LIN {X 0,Y 197.499,Z 678.187,A -85,B 0,C 180,E1 -21855.576,E2 -21855.576} C_VEL
LIN {X 0,Y 195.78,Z 682.074,A -85,B 0,C 180,E1 -21858.613,E2 -21858.613} C_VEL
LIN {X 0,Y 194.459,Z 684.943,A -85,B 0,C 180,E1 -21861.688,E2 -21861.688} C_VEL
LIN {X 0,Y 194.056,Z 686.281,A -85,B 0,C 180,E1 -21863.763,E2 -21863.763} C_VEL
LIN {X 0,Y 193.799,Z 687.228,A -85,B 0,C 180,E1 -21865.841,E2 -21865.841} C_VEL
LIN {X 0,Y 193.417,Z 688.055,A -85,B 0,C 180,E1 -21870,E2 -21870} C_VEL
LIN {X 0,Y 193.796,Z 687.282,A -85,B 0,C 180,E1 -21874.159,E2 -21874.159} C_VEL
LIN {X 0,Y 194.443,Z 685.054,A -85,B 0,C 180,E1 -21878.313,E2 -21878.313} C_VEL
LIN {X 0,Y 195.772,Z 682.224,A -85,B 0,C 180,E1 -21881.387,E2 -21881.387} C_VEL
LIN {X 0,Y 197.474,Z 678.391,A -85,B 0,C 180,E1 -21884.425,E2 -21884.425} C_VEL
LIN {X 0,Y 199.366,Z 673.305,A -85,B 0,C 180,E1 -21887.541,E2 -21887.541} C_VEL
LIN {X 0,Y 201.662,Z 667.266,A -85,B 0,C 180,E1 -21890.395,E2 -21890.395} C_VEL
LIN {X 0,Y 204.413,Z 659.477,A -85,B 0,C 180,E1 -21893.289,E2 -21893.289} C_VEL
LIN {X 0,Y 207.374,Z 649.797,A -85,B 0,C 180,E1 -21896.14,E2 -21896.14} C_VEL
LIN {X 0,Y 209.903,Z 640.74,A -85,B 0,C 180,E1 -21898.224,E2 -21898.224} C_VEL
LIN {X 0,Y 212.551,Z 630.212,A -85,B 0,C 180,E1 -21900.13,E2 -21900.13} C_VEL
LIN {X 0,Y 214.851,Z 618.67,A -85,B 0,C 180,E1 -21901.781,E2 -21901.781} C_VEL
LIN {X 0,Y 216.718,Z 607.358,A -85,B 0,C 180,E1 -21902.997,E2 -21902.997} C_VEL
LIN {X 0,Y 217.85,Z 594.616,A -85,B 0,C 180,E1 -21904.049,E2 -21904.049} C_VEL
LIN {X 0,Y 218.527,Z 581.541,A -85,B 0,C 180,E1 -21904.74,E2 -21904.74} C_VEL
LIN {X 0,Y 219.472,Z 546.637,A -85,B 0,C 180,E1 -21905.962,E2 -21905.962} C_VEL
LIN {X 0,Y 212.575,Z 532.953,A -85,B 0,C 180,E1 -21907.952,E2 -21907.952} C_VEL
LIN {X 0,Y 205.517,Z 520.799,A -85,B 0,C 180,E1 -21910.109,E2 -21910.109} C_VEL
LIN {X 0,Y 200.207,Z 512.651,A -85,B 0,C 180,E1 -21911.836,E2 -21911.836} C_VEL
LIN {X 0,Y 197.755,Z 509.046,A -85,B 0,C 180,E1 -21912.674,E2 -21912.674} C_VEL
LIN {X 0,Y 195.601,Z 505.666,A -85,B 0,C 180,E1 -21913.449,E2 -21913.449} C_VEL
LIN {X 0,Y 193.302,Z 502.912,A -85,B 0,C 180,E1 -21914.263,E2 -21914.263} C_VEL
LIN {X 0,Y 192.631,Z 500.948,A -85,B 0,C 180,E1 -21914.75,E2 -21914.75} C_VEL
LIN {X 0,Y 192.52,Z 500.498,A -85,B 0,C 180,E1 -21915.59,E2 -21915.59} C_VEL
LIN {X 0,Y 192.507,Z 500.453,A -85,B 0,C 180,E1 -21920.053,E2 -21920.053} C_VEL
LIN {X 0,Y 192.558,Z 500.5,A -85,B 0,C 180,E1 -21924.27,E2 -21924.27} C_VEL
LIN {X 0,Y 192.605,Z 500.44,A -85,B 0,C 180,E1 -21927.059,E2 -21927.059} C_VEL
LIN {X 0,Y 192.658,Z 500.435,A -85,B 0,C 180,E1 -21931.691,E2 -21931.691} C_VEL
LIN {X 0,Y 192.682,Z 500.469,A -85,B 0,C 180,E1 -21936.345,E2 -21936.345} C_VEL
LIN {X 0,Y 192.728,Z 500.474,A -85,B 0,C 180,E1 -21941.458,E2 -21941.458} C_VEL
LIN {X 0,Y 192.848,Z 500.463,A -85,B 0,C 180,E1 -21947.37,E2 -21947.37} C_VEL
LIN {X 0,Y 193.064,Z 500.413,A -85,B 0,C 180,E1 -21951.627,E2 -21951.627} C_VEL
LIN {X 0,Y 193.259,Z 500.383,A -85,B 0,C 180,E1 -21957.916,E2 -21957.916} C_VEL
LIN {X 0,Y 193.442,Z 500.381,A -85,B 0,C 180,E1 -21960,E2 -21960} C_VEL
LIN {X 0,Y 192.968,Z 500.419,A -85,B 0,C 180,E1 -21964.177,E2 -21964.177} C_VEL
LIN {X 0,Y 193.032,Z 500.437,A -85,B 0,C 180,E1 -21968.374,E2 -21968.374} C_VEL
LIN {X 0,Y 192.798,Z 500.454,A -85,B 0,C 180,E1 -21972.634,E2 -21972.634} C_VEL
LIN {X 0,Y 192.754,Z 500.439,A -85,B 0,C 180,E1 -21976.959,E2 -21976.959} C_VEL
LIN {X 0,Y 192.626,Z 500.465,A -85,B 0,C 180,E1 -21981.398,E2 -21981.398} C_VEL
LIN {X 0,Y 192.661,Z 500.476,A -85,B 0,C 180,E1 -21984.225,E2 -21984.225} C_VEL
LIN {X 0,Y 192.647,Z 500.468,A -85,B 0,C 180,E1 -21988.893,E2 -21988.893} C_VEL
LIN {X 0,Y 192.596,Z 500.469,A -85,B 0,C 180,E1 -21993.186,E2 -21993.186} C_VEL
LIN {X 0,Y 192.61,Z 500.721,A -85,B 0,C 180,E1 -21994.759,E2 -21994.759} C_VEL
LIN {X 0,Y 195.27,Z 509.211,A -85,B 0,C 180,E1 -21999.706,E2 -21999.706} C_VEL
LIN {X 0,Y 197.737,Z 517.882,A -85,B 0,C 180,E1 -22004.176,E2 -22004.176} C_VEL
LIN {X 0,Y 198.984,Z 522.474,A -85,B 0,C 180,E1 -22006.298,E2 -22006.298} C_VEL
LIN {X 0,Y 204.591,Z 534.212,A -85,B 0,C 180,E1 -22008.344,E2 -22008.344} C_VEL
LIN {X 0,Y 210.617,Z 548.053,A -85,B 0,C 180,E1 -22010.333,E2 -22010.333} C_VEL
LIN {X 0,Y 211.524,Z 550.943,A -85,B 0,C 180,E1 -22010.653,E2 -22010.653} C_VEL
LIN {X 0,Y 214.13,Z 576.298,A -85,B 0,C 180,E1 -22012.25,E2 -22012.25} C_VEL
LIN {X 0,Y 216.129,Z 604.791,A -85,B 0,C 180,E1 -22013.789,E2 -22013.789} C_VEL
LIN {X 0,Y 216.582,Z 612.878,A -85,B 0,C 180,E1 -22014.194,E2 -22014.194} C_VEL
LIN {X 0,Y 216.05,Z 618.711,A -85,B 0,C 180,E1 -22014.32,E2 -22014.32} C_VEL
LIN {X 0,Y 214.533,Z 624.449,A -85,B 0,C 180,E1 -22014.265,E2 -22014.265} C_VEL
LIN {X 0,Y 209.975,Z 637.636,A -85,B 0,C 180,E1 -22014.06,E2 -22014.06} C_VEL
LIN {X 0,Y 208.782,Z 643.411,A -85,B 0,C 180,E1 -22014.266,E2 -22014.266} C_VEL
LIN {X 0,Y 206.963,Z 656.057,A -85,B 0,C 180,E1 -22015.187,E2 -22015.187} C_VEL
LIN {X 0,Y 205.094,Z 665.781,A -85,B 0,C 180,E1 -22016.163,E2 -22016.163} C_VEL
LIN {X 0,Y 202.171,Z 677.646,A -85,B 0,C 180,E1 -22017.693,E2 -22017.693} C_VEL
LIN {X 0,Y 198.651,Z 689.501,A -85,B 0,C 180,E1 -22019.726,E2 -22019.726} C_VEL
LIN {X 0,Y 195.192,Z 700.074,A -85,B 0,C 180,E1 -22022.092,E2 -22022.092} C_VEL
LIN {X 0,Y 192.203,Z 708.672,A -85,B 0,C 180,E1 -22024.556,E2 -22024.556} C_VEL
LIN {X 0,Y 189.306,Z 717.125,A -85,B 0,C 180,E1 -22027.634,E2 -22027.634} C_VEL
LIN {X 0,Y 186.845,Z 723.957,A -85,B 0,C 180,E1 -22030.785,E2 -22030.785} C_VEL
LIN {X 0,Y 185.18,Z 730.323,A -85,B 0,C 180,E1 -22034.594,E2 -22034.594} C_VEL
LIN {X 0,Y 184.386,Z 734.512,A -85,B 0,C 180,E1 -22037.899,E2 -22037.899} C_VEL
LIN {X 0,Y 184.257,Z 737.676,A -85,B 0,C 180,E1 -22041.224,E2 -22041.224} C_VEL
LIN {X 0,Y 184.433,Z 739.217,A -85,B 0,C 180,E1 -22043.436,E2 -22043.436} C_VEL
LIN {X 0,Y 184.793,Z 740.348,A -85,B 0,C 180,E1 -22045.638,E2 -22045.638} C_VEL
LIN {X 0,Y 185.84,Z 741.38,A -85,B 0,C 180,E1 -22050,E2 -22050} C_VEL
LIN {X 0,Y 184.812,Z 740.331,A -85,B 0,C 180,E1 -22054.362,E2 -22054.362} C_VEL
LIN {X 0,Y 184.36,Z 738.485,A -85,B 0,C 180,E1 -22057.629,E2 -22057.629} C_VEL
LIN {X 0,Y 184.285,Z 735.608,A -85,B 0,C 180,E1 -22060.992,E2 -22060.992} C_VEL
LIN {X 0,Y 184.851,Z 731.751,A -85,B 0,C 180,E1 -22064.307,E2 -22064.307} C_VEL
LIN {X 0,Y 186.073,Z 726.793,A -85,B 0,C 180,E1 -22067.587,E2 -22067.587} C_VEL
LIN {X 0,Y 188.212,Z 720.14,A -85,B 0,C 180,E1 -22071.009,E2 -22071.009} C_VEL
LIN {X 0,Y 190.673,Z 712.967,A -85,B 0,C 180,E1 -22073.919,E2 -22073.919} C_VEL
LIN {X 0,Y 193.385,Z 705.23,A -85,B 0,C 180,E1 -22076.435,E2 -22076.435} C_VEL
LIN {X 0,Y 196.501,Z 695.896,A -85,B 0,C 180,E1 -22078.87,E2 -22078.87} C_VEL
LIN {X 0,Y 199.834,Z 685.58,A -85,B 0,C 180,E1 -22080.953,E2 -22080.953} C_VEL
LIN {X 0,Y 203.037,Z 674.165,A -85,B 0,C 180,E1 -22082.741,E2 -22082.741} C_VEL
LIN {X 0,Y 205.619,Z 662.301,A -85,B 0,C 180,E1 -22084.181,E2 -22084.181} C_VEL
LIN {X 0,Y 207.884,Z 649.433,A -85,B 0,C 180,E1 -22085.29,E2 -22085.29} C_VEL
LIN {X 0,Y 209.429,Z 635.954,A -85,B 0,C 180,E1 -22086.076,E2 -22086.076} C_VEL
LIN {X 0,Y 210.609,Z 611.893,A -85,B 0,C 180,E1 -22086.916,E2 -22086.916} C_VEL
LIN {X 0,Y 208.307,Z 576.822,A -85,B 0,C 180,E1 -22088.861,E2 -22088.861} C_VEL
LIN {X 0,Y 205.939,Z 552.664,A -85,B 0,C 180,E1 -22090.435,E2 -22090.435} C_VEL
LIN {X 0,Y 201.062,Z 541.037,A -85,B 0,C 180,E1 -22092.124,E2 -22092.124} C_VEL
LIN {X 0,Y 196.044,Z 530.426,A -85,B 0,C 180,E1 -22093.935,E2 -22093.935} C_VEL
LIN {X 0,Y 193.42,Z 525.344,A -85,B 0,C 180,E1 -22094.918,E2 -22094.918} C_VEL
LIN {X 0,Y 191.371,Z 520.955,A -85,B 0,C 180,E1 -22095.844,E2 -22095.844} C_VEL
LIN {X 0,Y 189.045,Z 512.792,A -85,B 0,C 180,E1 -22100.112,E2 -22100.112} C_VEL
LIN {X 0,Y 186.806,Z 505.66,A -85,B 0,C 180,E1 -22104.328,E2 -22104.328} C_VEL
LIN {X 0,Y 185.567,Z 501.428,A -85,B 0,C 180,E1 -22107.137,E2 -22107.137} C_VEL
LIN {X 0,Y 185.579,Z 501.355,A -85,B 0,C 180,E1 -22110.575,E2 -22110.575} C_VEL
LIN {X 0,Y 185.584,Z 501.35,A -85,B 0,C 180,E1 -22115.382,E2 -22115.382} C_VEL
LIN {X 0,Y 185.67,Z 501.308,A -85,B 0,C 180,E1 -22121.134,E2 -22121.134} C_VEL
LIN {X 0,Y 185.691,Z 501.349,A -85,B 0,C 180,E1 -22124.637,E2 -22124.637} C_VEL
LIN {X 0,Y 185.885,Z 501.307,A -85,B 0,C 180,E1 -22129.418,E2 -22129.418} C_VEL
LIN {X 0,Y 185.944,Z 501.313,A -85,B 0,C 180,E1 -22133.489,E2 -22133.489} C_VEL
LIN {X 0,Y 186.202,Z 501.28,A -85,B 0,C 180,E1 -22137.837,E2 -22137.837} C_VEL
LIN {X 0,Y 186.405,Z 501.261,A -85,B 0,C 180,E1 -22140,E2 -22140} C_VEL
LIN {X 0,Y 185.916,Z 501.309,A -85,B 0,C 180,E1 -22144.336,E2 -22144.336} C_VEL
LIN {X 0,Y 185.979,Z 501.293,A -85,B 0,C 180,E1 -22148.694,E2 -22148.694} C_VEL
LIN {X 0,Y 185.724,Z 501.35,A -85,B 0,C 180,E1 -22153.123,E2 -22153.123} C_VEL
LIN {X 0,Y 185.685,Z 501.339,A -85,B 0,C 180,E1 -22157.626,E2 -22157.626} C_VEL
LIN {X 0,Y 185.577,Z 501.347,A -85,B 0,C 180,E1 -22162.254,E2 -22162.254} C_VEL
LIN {X 0,Y 185.556,Z 501.345,A -85,B 0,C 180,E1 -22167.033,E2 -22167.033} C_VEL
LIN {X 0,Y 185.575,Z 501.3,A -85,B 0,C 180,E1 -22169.494,E2 -22169.494} C_VEL
LIN {X 0,Y 185.496,Z 501.359,A -85,B 0,C 180,E1 -22174.633,E2 -22174.633} C_VEL
LIN {X 0,Y 185.499,Z 501.35,A -85,B 0,C 180,E1 -22177.315,E2 -22177.315} C_VEL
LIN {X 0,Y 185.469,Z 501.445,A -85,B 0,C 180,E1 -22182.771,E2 -22182.771} C_VEL
LIN {X 0,Y 185.629,Z 502.258,A -85,B 0,C 180,E1 -22183.39,E2 -22183.39} C_VEL
LIN {X 0,Y 187.124,Z 505.129,A -85,B 0,C 180,E1 -22184.12,E2 -22184.12} C_VEL
LIN {X 0,Y 188.874,Z 506.941,A -85,B 0,C 180,E1 -22184.781,E2 -22184.781} C_VEL
LIN {X 0,Y 190.87,Z 510.07,A -85,B 0,C 180,E1 -22185.568,E2 -22185.568} C_VEL
LIN {X 0,Y 192.372,Z 512.165,A -85,B 0,C 180,E1 -22186.129,E2 -22186.129} C_VEL
LIN {X 0,Y 197.664,Z 519.995,A -85,B 0,C 180,E1 -22188.019,E2 -22188.019} C_VEL
LIN {X 0,Y 203.928,Z 530.25,A -85,B 0,C 180,E1 -22190.108,E2 -22190.108} C_VEL
LIN {X 0,Y 211.258,Z 543.831,A -85,B 0,C 180,E1 -22192.39,E2 -22192.39} C_VEL
LIN {X 0,Y 213.706,Z 549.024,A -85,B 0,C 180,E1 -22193.13,E2 -22193.13} C_VEL
LIN {X 0,Y 212.454,Z 587.486,A -85,B 0,C 180,E1 -22194.541,E2 -22194.541} C_VEL
LIN {X 0,Y 211.413,Z 601.314,A -85,B 0,C 180,E1 -22195.451,E2 -22195.451} C_VEL
LIN {X 0,Y 209.843,Z 613.54,A -85,B 0,C 180,E1 -22196.614,E2 -22196.614} C_VEL
LIN {X 0,Y 207.843,Z 624.696,A -85,B 0,C 180,E1 -22198.032,E2 -22198.032} C_VEL
LIN {X 0,Y 205.358,Z 635.064,A -85,B 0,C 180,E1 -22199.683,E2 -22199.683} C_VEL
LIN {X 0,Y 202.579,Z 645.376,A -85,B 0,C 180,E1 -22201.792,E2 -22201.792} C_VEL
LIN {X 0,Y 200.031,Z 653.784,A -85,B 0,C 180,E1 -22203.949,E2 -22203.949} C_VEL
LIN {X 0,Y 197.499,Z 661.508,A -85,B 0,C 180,E1 -22206.402,E2 -22206.402} C_VEL
LIN {X 0,Y 194.636,Z 669.172,A -85,B 0,C 180,E1 -22209.443,E2 -22209.443} C_VEL
LIN {X 0,Y 191.978,Z 675.971,A -85,B 0,C 180,E1 -22212.971,E2 -22212.971} C_VEL
LIN {X 0,Y 190.005,Z 680.577,A -85,B 0,C 180,E1 -22216.089,E2 -22216.089} C_VEL
LIN {X 0,Y 188.343,Z 684.112,A -85,B 0,C 180,E1 -22219.247,E2 -22219.247} C_VEL
LIN {X 0,Y 187.506,Z 685.933,A -85,B 0,C 180,E1 -22221.378,E2 -22221.378} C_VEL
LIN {X 0,Y 187.07,Z 687.27,A -85,B 0,C 180,E1 -22223.529,E2 -22223.529} C_VEL
LIN {X 0,Y 186.791,Z 688.216,A -85,B 0,C 180,E1 -22225.685,E2 -22225.685} C_VEL
LIN {X 0,Y 186.389,Z 689.043,A -85,B 0,C 180,E1 -22230,E2 -22230} C_VEL
LIN {X 0,Y 186.788,Z 688.269,A -85,B 0,C 180,E1 -22234.316,E2 -22234.316} C_VEL
LIN {X 0,Y 187.489,Z 686.042,A -85,B 0,C 180,E1 -22238.623,E2 -22238.623} C_VEL
LIN {X 0,Y 188.888,Z 683.211,A -85,B 0,C 180,E1 -22241.808,E2 -22241.808} C_VEL
LIN {X 0,Y 190.676,Z 679.378,A -85,B 0,C 180,E1 -22244.952,E2 -22244.952} C_VEL
LIN {X 0,Y 192.676,Z 674.291,A -85,B 0,C 180,E1 -22248.171,E2 -22248.171} C_VEL
LIN {X 0,Y 195.09,Z 668.252,A -85,B 0,C 180,E1 -22251.115,E2 -22251.115} C_VEL
LIN {X 0,Y 197.977,Z 660.463,A -85,B 0,C 180,E1 -22254.094,E2 -22254.094} C_VEL
LIN {X 0,Y 201.088,Z 650.782,A -85,B 0,C 180,E1 -22257.022,E2 -22257.022} C_VEL
LIN {X 0,Y 203.74,Z 641.724,A -85,B 0,C 180,E1 -22259.159,E2 -22259.159} C_VEL
LIN {X 0,Y 206.51,Z 631.193,A -85,B 0,C 180,E1 -22261.107,E2 -22261.107} C_VEL
LIN {X 0,Y 208.95,Z 619.496,A -85,B 0,C 180,E1 -22262.815,E2 -22262.815} C_VEL
LIN {X 0,Y 210.905,Z 607.994,A -85,B 0,C 180,E1 -22264.071,E2 -22264.071} C_VEL
LIN {X 0,Y 212.098,Z 595.07,A -85,B 0,C 180,E1 -22265.148,E2 -22265.148} C_VEL
LIN {X 0,Y 212.79,Z 581.576,A -85,B 0,C 180,E1 -22265.865,E2 -22265.865} C_VEL
LIN {X 0,Y 213.713,Z 548.894,A -85,B 0,C 180,E1 -22267.038,E2 -22267.038} C_VEL
LIN {X 0,Y 207.503,Z 536.628,A -85,B 0,C 180,E1 -22268.93,E2 -22268.93} C_VEL
LIN {X 0,Y 201.238,Z 525.581,A -85,B 0,C 180,E1 -22270.954,E2 -22270.954} C_VEL
LIN {X 0,Y 194.118,Z 514.597,A -85,B 0,C 180,E1 -22273.425,E2 -22273.425} C_VEL
LIN {X 0,Y 190.785,Z 509.938,A -85,B 0,C 180,E1 -22274.658,E2 -22274.658} C_VEL
LIN {X 0,Y 188.759,Z 506.737,A -85,B 0,C 180,E1 -22275.463,E2 -22275.463} C_VEL
LIN {X 0,Y 186.229,Z 503.818,A -85,B 0,C 180,E1 -22276.45,E2 -22276.45} C_VEL
LIN {X 0,Y 185.573,Z 501.969,A -85,B 0,C 180,E1 -22276.928,E2 -22276.928} C_VEL
LIN {X 0,Y 185.46,Z 501.409,A -85,B 0,C 180,E1 -22277.617,E2 -22277.617} C_VEL
LIN {X 0,Y 185.5,Z 501.349,A -85,B 0,C 180,E1 -22282.712,E2 -22282.712} C_VEL
LIN {X 0,Y 185.539,Z 501.306,A -85,B 0,C 180,E1 -22287.974,E2 -22287.974} C_VEL
LIN {X 0,Y 185.578,Z 501.301,A -85,B 0,C 180,E1 -22290.576,E2 -22290.576} C_VEL
LIN {X 0,Y 185.577,Z 501.365,A -85,B 0,C 180,E1 -22295.381,E2 -22295.381} C_VEL
LIN {X 0,Y 185.671,Z 501.356,A -85,B 0,C 180,E1 -22301.134,E2 -22301.134} C_VEL
LIN {X 0,Y 185.759,Z 501.346,A -85,B 0,C 180,E1 -22306.879,E2 -22306.879} C_VEL
LIN {X 0,Y 186.01,Z 501.289,A -85,B 0,C 180,E1 -22311.307,E2 -22311.307} C_VEL
LIN {X 0,Y 186.203,Z 501.261,A -85,B 0,C 180,E1 -22317.837,E2 -22317.837} C_VEL
LIN {X 0,Y 186.405,Z 501.257,A -85,B 0,C 180,E1 -22320,E2 -22320} C_VEL
LIN {X 0,Y 185.915,Z 501.297,A -85,B 0,C 180,E1 -22324.336,E2 -22324.336} C_VEL
LIN {X 0,Y 185.979,Z 501.31,A -85,B 0,C 180,E1 -22328.694,E2 -22328.694} C_VEL
LIN {X 0,Y 185.725,Z 501.341,A -85,B 0,C 180,E1 -22333.123,E2 -22333.123} C_VEL
LIN {X 0,Y 185.686,Z 501.311,A -85,B 0,C 180,E1 -22337.625,E2 -22337.625} C_VEL
LIN {X 0,Y 185.59,Z 501.358,A -85,B 0,C 180,E1 -22342.252,E2 -22342.252} C_VEL
LIN {X 0,Y 185.559,Z 501.335,A -85,B 0,C 180,E1 -22347.033,E2 -22347.033} C_VEL
LIN {X 0,Y 185.576,Z 501.358,A -85,B 0,C 180,E1 -22349.494,E2 -22349.494} C_VEL
LIN {X 0,Y 185.603,Z 501.511,A -85,B 0,C 180,E1 -22352.888,E2 -22352.888} C_VEL
LIN {X 0,Y 188.362,Z 510.35,A -85,B 0,C 180,E1 -22358.417,E2 -22358.417} C_VEL
LIN {X 0,Y 190.741,Z 518.676,A -85,B 0,C 180,E1 -22362.975,E2 -22362.975} C_VEL
LIN {X 0,Y 191.435,Z 521.22,A -85,B 0,C 180,E1 -22364.138,E2 -22364.138} C_VEL
LIN {X 0,Y 195.498,Z 529.272,A -85,B 0,C 180,E1 -22365.767,E2 -22365.767} C_VEL
LIN {X 0,Y 200.116,Z 538.807,A -85,B 0,C 180,E1 -22367.449,E2 -22367.449} C_VEL
LIN {X 0,Y 205.59,Z 551.566,A -85,B 0,C 180,E1 -22369.358,E2 -22369.358} C_VEL
LIN {X 0,Y 206.205,Z 554.163,A -85,B 0,C 180,E1 -22369.615,E2 -22369.615} C_VEL
LIN {X 0,Y 208.646,Z 579.601,A -85,B 0,C 180,E1 -22371.257,E2 -22371.257} C_VEL
LIN {X 0,Y 210.719,Z 611.4,A -85,B 0,C 180,E1 -22373.016,E2 -22373.016} C_VEL
LIN {X 0,Y 209.623,Z 634.88,A -85,B 0,C 180,E1 -22373.824,E2 -22373.824} C_VEL
LIN {X 0,Y 208.782,Z 643.411,A -85,B 0,C 180,E1 -22374.266,E2 -22374.266} C_VEL
LIN {X 0,Y 207.502,Z 649.097,A -85,B 0,C 180,E1 -22374.532,E2 -22374.532} C_VEL
LIN {X 0,Y 203.648,Z 658.159,A -85,B 0,C 180,E1 -22374.851,E2 -22374.851} C_VEL
LIN {X 0,Y 199.388,Z 666.921,A -85,B 0,C 180,E1 -22375.368,E2 -22375.368} C_VEL
LIN {X 0,Y 197.488,Z 672.139,A -85,B 0,C 180,E1 -22375.949,E2 -22375.949} C_VEL
LIN {X 0,Y 194.138,Z 683.569,A -85,B 0,C 180,E1 -22377.727,E2 -22377.727} C_VEL
LIN {X 0,Y 190.672,Z 694.076,A -85,B 0,C 180,E1 -22379.855,E2 -22379.855} C_VEL
LIN {X 0,Y 187.618,Z 702.705,A -85,B 0,C 180,E1 -22382.081,E2 -22382.081} C_VEL
LIN {X 0,Y 184.689,Z 710.708,A -85,B 0,C 180,E1 -22384.654,E2 -22384.654} C_VEL
LIN {X 0,Y 181.809,Z 718.61,A -85,B 0,C 180,E1 -22387.876,E2 -22387.876} C_VEL
LIN {X 0,Y 179.783,Z 723.985,A -85,B 0,C 180,E1 -22390.593,E2 -22390.593} C_VEL
LIN {X 0,Y 178.284,Z 729.317,A -85,B 0,C 180,E1 -22393.982,E2 -22393.982} C_VEL
LIN {X 0,Y 177.383,Z 733.505,A -85,B 0,C 180,E1 -22397.414,E2 -22397.414} C_VEL
LIN {X 0,Y 177.203,Z 736.673,A -85,B 0,C 180,E1 -22400.872,E2 -22400.872} C_VEL
LIN {X 0,Y 177.356,Z 738.215,A -85,B 0,C 180,E1 -22403.173,E2 -22403.173} C_VEL
LIN {X 0,Y 177.703,Z 739.348,A -85,B 0,C 180,E1 -22405.463,E2 -22405.463} C_VEL
LIN {X 0,Y 178.789,Z 740.389,A -85,B 0,C 180,E1 -22410,E2 -22410} C_VEL
LIN {X 0,Y 177.721,Z 739.331,A -85,B 0,C 180,E1 -22414.536,E2 -22414.536} C_VEL
LIN {X 0,Y 177.286,Z 737.664,A -85,B 0,C 180,E1 -22417.67,E2 -22417.67} C_VEL
LIN {X 0,Y 177.265,Z 734.601,A -85,B 0,C 180,E1 -22421.433,E2 -22421.433} C_VEL
LIN {X 0,Y 177.906,Z 730.741,A -85,B 0,C 180,E1 -22424.878,E2 -22424.878} C_VEL
LIN {X 0,Y 179.241,Z 725.782,A -85,B 0,C 180,E1 -22428.281,E2 -22428.281} C_VEL
LIN {X 0,Y 181.37,Z 719.664,A -85,B 0,C 180,E1 -22431.567,E2 -22431.567} C_VEL
LIN {X 0,Y 184.153,Z 711.958,A -85,B 0,C 180,E1 -22434.822,E2 -22434.822} C_VEL
LIN {X 0,Y 187.016,Z 704.223,A -85,B 0,C 180,E1 -22437.409,E2 -22437.409} C_VEL
LIN {X 0,Y 190.307,Z 694.894,A -85,B 0,C 180,E1 -22439.903,E2 -22439.903} C_VEL
LIN {X 0,Y 193.787,Z 684.579,A -85,B 0,C 180,E1 -22442.032,E2 -22442.032} C_VEL
LIN {X 0,Y 197.099,Z 673.161,A -85,B 0,C 180,E1 -22443.858,E2 -22443.858} C_VEL
LIN {X 0,Y 199.741,Z 661.289,A -85,B 0,C 180,E1 -22445.334,E2 -22445.334} C_VEL
LIN {X 0,Y 202.108,Z 648.568,A -85,B 0,C 180,E1 -22446.443,E2 -22446.443} C_VEL
LIN {X 0,Y 203.614,Z 636.122,A -85,B 0,C 180,E1 -22447.197,E2 -22447.197} C_VEL
LIN {X 0,Y 204.903,Z 615.139,A -85,B 0,C 180,E1 -22447.94,E2 -22447.94} C_VEL
LIN {X 0,Y 203.278,Z 585.097,A -85,B 0,C 180,E1 -22449.603,E2 -22449.603} C_VEL
LIN {X 0,Y 200.708,Z 555.786,A -85,B 0,C 180,E1 -22451.529,E2 -22451.529} C_VEL
LIN {X 0,Y 197.732,Z 548.261,A -85,B 0,C 180,E1 -22452.627,E2 -22452.627} C_VEL
LIN {X 0,Y 192.465,Z 536.379,A -85,B 0,C 180,E1 -22454.633,E2 -22454.633} C_VEL
LIN {X 0,Y 188.757,Z 529.157,A -85,B 0,C 180,E1 -22456.095,E2 -22456.095} C_VEL
LIN {X 0,Y 186.274,Z 524.432,A -85,B 0,C 180,E1 -22457.123,E2 -22457.123} C_VEL
LIN {X 0,Y 183.734,Z 519.425,A -85,B 0,C 180,E1 -22458.348,E2 -22458.348} C_VEL
LIN {X 0,Y 181.965,Z 513.227,A -85,B 0,C 180,E1 -22461.832,E2 -22461.832} C_VEL
LIN {X 0,Y 179.496,Z 505.59,A -85,B 0,C 180,E1 -22466.759,E2 -22466.759} C_VEL
LIN {X 0,Y 178.49,Z 502.306,A -85,B 0,C 180,E1 -22469.211,E2 -22469.211} C_VEL
LIN {X 0,Y 178.503,Z 502.219,A -85,B 0,C 180,E1 -22474.336,E2 -22474.336} C_VEL
LIN {X 0,Y 178.526,Z 502.208,A -85,B 0,C 180,E1 -22479.249,E2 -22479.249} C_VEL
LIN {X 0,Y 178.646,Z 502.183,A -85,B 0,C 180,E1 -22481.656,E2 -22481.656} C_VEL
LIN {X 0,Y 178.654,Z 502.228,A -85,B 0,C 180,E1 -22486.348,E2 -22486.348} C_VEL
LIN {X 0,Y 178.908,Z 502.189,A -85,B 0,C 180,E1 -22490.96,E2 -22490.96} C_VEL
LIN {X 0,Y 179.148,Z 502.157,A -85,B 0,C 180,E1 -22497.752,E2 -22497.752} C_VEL
LIN {X 0,Y 179.368,Z 502.137,A -85,B 0,C 180,E1 -22500,E2 -22500} C_VEL
LIN {X 0,Y 178.864,Z 502.189,A -85,B 0,C 180,E1 -22504.507,E2 -22504.507} C_VEL
LIN {X 0,Y 178.908,Z 502.172,A -85,B 0,C 180,E1 -22509.041,E2 -22509.041} C_VEL
LIN {X 0,Y 178.652,Z 502.226,A -85,B 0,C 180,E1 -22513.653,E2 -22513.653} C_VEL
LIN {X 0,Y 178.619,Z 502.237,A -85,B 0,C 180,E1 -22519.215,E2 -22519.215} C_VEL
LIN {X 0,Y 178.517,Z 502.248,A -85,B 0,C 180,E1 -22525.115,E2 -22525.115} C_VEL
LIN {X 0,Y 178.519,Z 502.175,A -85,B 0,C 180,E1 -22529.993,E2 -22529.993} C_VEL
LIN {X 0,Y 178.482,Z 502.219,A -85,B 0,C 180,E1 -22534.22,E2 -22534.22} C_VEL
LIN {X 0,Y 178.449,Z 502.268,A -85,B 0,C 180,E1 -22540.159,E2 -22540.159} C_VEL
LIN {X 0,Y 178.595,Z 503.083,A -85,B 0,C 180,E1 -22540.898,E2 -22540.898} C_VEL
LIN {X 0,Y 179.978,Z 505.859,A -85,B 0,C 180,E1 -22541.674,E2 -22541.674} C_VEL
LIN {X 0,Y 181.907,Z 507.76,A -85,B 0,C 180,E1 -22542.488,E2 -22542.488} C_VEL
LIN {X 0,Y 183.903,Z 510.97,A -85,B 0,C 180,E1 -22543.369,E2 -22543.369} C_VEL
LIN {X 0,Y 185.419,Z 512.873,A -85,B 0,C 180,E1 -22543.986,E2 -22543.986} C_VEL
LIN {X 0,Y 189.076,Z 518.203,A -85,B 0,C 180,E1 -22545.447,E2 -22545.447} C_VEL
LIN {X 0,Y 194.236,Z 525.984,A -85,B 0,C 180,E1 -22547.369,E2 -22547.369} C_VEL
LIN {X 0,Y 201.142,Z 537.653,A -85,B 0,C 180,E1 -22549.763,E2 -22549.763} C_VEL
LIN {X 0,Y 207.965,Z 551.175,A -85,B 0,C 180,E1 -22551.982,E2 -22551.982} C_VEL
LIN {X 0,Y 206.764,Z 588.816,A -85,B 0,C 180,E1 -22553.432,E2 -22553.432} C_VEL
LIN {X 0,Y 205.658,Z 602.389,A -85,B 0,C 180,E1 -22554.347,E2 -22554.347} C_VEL
LIN {X 0,Y 204.011,Z 614.535,A -85,B 0,C 180,E1 -22555.527,E2 -22555.527} C_VEL
LIN {X 0,Y 201.916,Z 625.684,A -85,B 0,C 180,E1 -22556.976,E2 -22556.976} C_VEL
LIN {X 0,Y 199.324,Z 636.056,A -85,B 0,C 180,E1 -22558.664,E2 -22558.664} C_VEL
LIN {X 0,Y 196.413,Z 646.368,A -85,B 0,C 180,E1 -22560.823,E2 -22560.823} C_VEL
LIN {X 0,Y 193.741,Z 654.775,A -85,B 0,C 180,E1 -22563.036,E2 -22563.036} C_VEL
LIN {X 0,Y 191.079,Z 662.498,A -85,B 0,C 180,E1 -22565.558,E2 -22565.558} C_VEL
LIN {X 0,Y 188.071,Z 670.162,A -85,B 0,C 180,E1 -22568.691,E2 -22568.691} C_VEL
LIN {X 0,Y 185.269,Z 676.96,A -85,B 0,C 180,E1 -22572.334,E2 -22572.334} C_VEL
LIN {X 0,Y 183.19,Z 681.566,A -85,B 0,C 180,E1 -22575.56,E2 -22575.56} C_VEL
LIN {X 0,Y 181.441,Z 685.101,A -85,B 0,C 180,E1 -22578.833,E2 -22578.833} C_VEL
LIN {X 0,Y 180.558,Z 686.922,A -85,B 0,C 180,E1 -22581.043,E2 -22581.043} C_VEL
LIN {X 0,Y 180.088,Z 688.259,A -85,B 0,C 180,E1 -22583.277,E2 -22583.277} C_VEL
LIN {X 0,Y 179.785,Z 689.205,A -85,B 0,C 180,E1 -22585.516,E2 -22585.516} C_VEL
LIN {X 0,Y 179.361,Z 690.031,A -85,B 0,C 180,E1 -22590,E2 -22590} C_VEL
LIN {X 0,Y 179.781,Z 689.257,A -85,B 0,C 180,E1 -22594.484,E2 -22594.484} C_VEL
LIN {X 0,Y 180.541,Z 687.03,A -85,B 0,C 180,E1 -22598.958,E2 -22598.958} C_VEL
LIN {X 0,Y 182.014,Z 684.198,A -85,B 0,C 180,E1 -22602.261,E2 -22602.261} C_VEL
LIN {X 0,Y 183.894,Z 680.365,A -85,B 0,C 180,E1 -22605.517,E2 -22605.517} C_VEL
LIN {X 0,Y 186.012,Z 675.278,A -85,B 0,C 180,E1 -22608.846,E2 -22608.846} C_VEL
LIN {X 0,Y 188.551,Z 669.238,A -85,B 0,C 180,E1 -22611.884,E2 -22611.884} C_VEL
LIN {X 0,Y 191.582,Z 661.449,A -85,B 0,C 180,E1 -22614.952,E2 -22614.952} C_VEL
LIN {X 0,Y 194.852,Z 651.767,A -85,B 0,C 180,E1 -22617.962,E2 -22617.962} C_VEL
LIN {X 0,Y 197.634,Z 642.708,A -85,B 0,C 180,E1 -22620.151,E2 -22620.151} C_VEL
LIN {X 0,Y 200.526,Z 632.177,A -85,B 0,C 180,E1 -22622.145,E2 -22622.145} C_VEL
LIN {X 0,Y 203.078,Z 620.478,A -85,B 0,C 180,E1 -22623.889,E2 -22623.889} C_VEL
LIN {X 0,Y 205.118,Z 608.975,A -85,B 0,C 180,E1 -22625.172,E2 -22625.172} C_VEL
LIN {X 0,Y 206.345,Z 596.586,A -85,B 0,C 180,E1 -22626.235,E2 -22626.235} C_VEL
LIN {X 0,Y 207.097,Z 585.021,A -85,B 0,C 180,E1 -22626.885,E2 -22626.885} C_VEL
LIN {X 0,Y 208.152,Z 551.453,A -85,B 0,C 180,E1 -22628.132,E2 -22628.132} C_VEL
LIN {X 0,Y 200.739,Z 536.928,A -85,B 0,C 180,E1 -22630.549,E2 -22630.549} C_VEL
LIN {X 0,Y 194.69,Z 526.671,A -85,B 0,C 180,E1 -22632.655,E2 -22632.655} C_VEL
LIN {X 0,Y 189.51,Z 518.84,A -85,B 0,C 180,E1 -22634.58,E2 -22634.58} C_VEL
LIN {X 0,Y 186.775,Z 514.917,A -85,B 0,C 180,E1 -22635.656,E2 -22635.656} C_VEL
LIN {X 0,Y 184.471,Z 511.572,A -85,B 0,C 180,E1 -22636.608,E2 -22636.608} C_VEL
LIN {X 0,Y 182.248,Z 508.496,A -85,B 0,C 180,E1 -22637.557,E2 -22637.557} C_VEL
LIN {X 0,Y 181.489,Z 507.27,A -85,B 0,C 180,E1 -22637.901,E2 -22637.901} C_VEL
LIN {X 0,Y 179.254,Z 504.796,A -85,B 0,C 180,E1 -22638.876,E2 -22638.876} C_VEL
LIN {X 0,Y 178.513,Z 502.73,A -85,B 0,C 180,E1 -22639.488,E2 -22639.488} C_VEL
LIN {X 0,Y 178.402,Z 502.26,A -85,B 0,C 180,E1 -22640.196,E2 -22640.196} C_VEL
LIN {X 0,Y 178.482,Z 502.22,A -85,B 0,C 180,E1 -22645.78,E2 -22645.78} C_VEL
LIN {X 0,Y 178.519,Z 502.175,A -85,B 0,C 180,E1 -22650.007,E2 -22650.007} C_VEL
LIN {X 0,Y 178.517,Z 502.249,A -85,B 0,C 180,E1 -22654.885,E2 -22654.885} C_VEL
LIN {X 0,Y 178.619,Z 502.236,A -85,B 0,C 180,E1 -22660.785,E2 -22660.785} C_VEL
LIN {X 0,Y 178.676,Z 502.224,A -85,B 0,C 180,E1 -22666.349,E2 -22666.349} C_VEL
LIN {X 0,Y 178.959,Z 502.165,A -85,B 0,C 180,E1 -22670.962,E2 -22670.962} C_VEL
LIN {X 0,Y 179.149,Z 502.139,A -85,B 0,C 180,E1 -22677.752,E2 -22677.752} C_VEL
LIN {X 0,Y 179.368,Z 502.133,A -85,B 0,C 180,E1 -22680,E2 -22680} C_VEL
LIN {X 0,Y 178.862,Z 502.176,A -85,B 0,C 180,E1 -22684.507,E2 -22684.507} C_VEL
LIN {X 0,Y 178.908,Z 502.186,A -85,B 0,C 180,E1 -22689.04,E2 -22689.04} C_VEL
LIN {X 0,Y 178.654,Z 502.228,A -85,B 0,C 180,E1 -22693.652,E2 -22693.652} C_VEL
LIN {X 0,Y 178.619,Z 502.186,A -85,B 0,C 180,E1 -22699.215,E2 -22699.215} C_VEL
LIN {X 0,Y 178.522,Z 502.221,A -85,B 0,C 180,E1 -22705.118,E2 -22705.118} C_VEL
LIN {X 0,Y 178.496,Z 502.299,A -85,B 0,C 180,E1 -22710.661,E2 -22710.661} C_VEL
LIN {X 0,Y 180.464,Z 508.589,A -85,B 0,C 180,E1 -22715.134,E2 -22715.134} C_VEL
LIN {X 0,Y 182.758,Z 516.056,A -85,B 0,C 180,E1 -22719.728,E2 -22719.728} C_VEL
LIN {X 0,Y 183.809,Z 519.685,A -85,B 0,C 180,E1 -22721.632,E2 -22721.632} C_VEL
LIN {X 0,Y 188.118,Z 527.839,A -85,B 0,C 180,E1 -22723.537,E2 -22723.537} C_VEL
LIN {X 0,Y 191.175,Z 533.763,A -85,B 0,C 180,E1 -22724.766,E2 -22724.766} C_VEL
LIN {X 0,Y 195.78,Z 543.605,A -85,B 0,C 180,E1 -22726.547,E2 -22726.547} C_VEL
LIN {X 0,Y 200.74,Z 555.463,A -85,B 0,C 180,E1 -22728.381,E2 -22728.381} C_VEL
LIN {X 0,Y 203.014,Z 580.05,A -85,B 0,C 180,E1 -22730.034,E2 -22730.034} C_VEL
LIN {X 0,Y 204.723,Z 607.61,A -85,B 0,C 180,E1 -22731.622,E2 -22731.622} C_VEL
LIN {X 0,Y 204.952,Z 616.236,A -85,B 0,C 180,E1 -22732.043,E2 -22732.043} C_VEL
LIN {X 0,Y 203.695,Z 636.301,A -85,B 0,C 180,E1 -22732.758,E2 -22732.758} C_VEL
LIN {X 0,Y 202.024,Z 649.874,A -85,B 0,C 180,E1 -22733.598,E2 -22733.598} C_VEL
LIN {X 0,Y 199.576,Z 662.775,A -85,B 0,C 180,E1 -22734.787,E2 -22734.787} C_VEL
LIN {X 0,Y 197.488,Z 672.139,A -85,B 0,C 180,E1 -22735.949,E2 -22735.949} C_VEL
LIN {X 0,Y 195.458,Z 677.349,A -85,B 0,C 180,E1 -22736.607,E2 -22736.607} C_VEL
LIN {X 0,Y 190.427,Z 685.341,A -85,B 0,C 180,E1 -22737.57,E2 -22737.57} C_VEL
LIN {X 0,Y 185.256,Z 692.749,A -85,B 0,C 180,E1 -22738.753,E2 -22738.753} C_VEL
LIN {X 0,Y 183.031,Z 697.091,A -85,B 0,C 180,E1 -22739.74,E2 -22739.74} C_VEL
LIN {X 0,Y 179.415,Z 706.669,A -85,B 0,C 180,E1 -22742.596,E2 -22742.596} C_VEL
LIN {X 0,Y 176.145,Z 715.115,A -85,B 0,C 180,E1 -22745.861,E2 -22745.861} C_VEL
LIN {X 0,Y 173.778,Z 720.903,A -85,B 0,C 180,E1 -22748.656,E2 -22748.656} C_VEL
LIN {X 0,Y 171.869,Z 726.642,A -85,B 0,C 180,E1 -22752.141,E2 -22752.141} C_VEL
LIN {X 0,Y 170.661,Z 731.201,A -85,B 0,C 180,E1 -22755.695,E2 -22755.695} C_VEL
LIN {X 0,Y 170.141,Z 734.696,A -85,B 0,C 180,E1 -22759.288,E2 -22759.288} C_VEL
LIN {X 0,Y 170.286,Z 737.214,A -85,B 0,C 180,E1 -22762.888,E2 -22762.888} C_VEL
LIN {X 0,Y 170.616,Z 738.349,A -85,B 0,C 180,E1 -22765.275,E2 -22765.275} C_VEL
LIN {X 0,Y 171.709,Z 739.393,A -85,B 0,C 180,E1 -22770,E2 -22770} C_VEL
LIN {X 0,Y 170.634,Z 738.331,A -85,B 0,C 180,E1 -22774.725,E2 -22774.725} C_VEL
LIN {X 0,Y 170.225,Z 736.825,A -85,B 0,C 180,E1 -22777.743,E2 -22777.743} C_VEL
LIN {X 0,Y 170.232,Z 733.59,A -85,B 0,C 180,E1 -22781.913,E2 -22781.913} C_VEL
LIN {X 0,Y 170.995,Z 729.733,A -85,B 0,C 180,E1 -22785.495,E2 -22785.495} C_VEL
LIN {X 0,Y 172.445,Z 724.772,A -85,B 0,C 180,E1 -22789.028,E2 -22789.028} C_VEL
LIN {X 0,Y 175.077,Z 717.772,A -85,B 0,C 180,E1 -22792.862,E2 -22792.862} C_VEL
LIN {X 0,Y 178.234,Z 709.529,A -85,B 0,C 180,E1 -22796.333,E2 -22796.333} C_VEL
LIN {X 0,Y 182.053,Z 699.689,A -85,B 0,C 180,E1 -22799.485,E2 -22799.485} C_VEL
LIN {X 0,Y 185.707,Z 689.575,A -85,B 0,C 180,E1 -22801.993,E2 -22801.993} C_VEL
LIN {X 0,Y 189.036,Z 679.627,A -85,B 0,C 180,E1 -22803.894,E2 -22803.894} C_VEL
LIN {X 0,Y 192.079,Z 668.827,A -85,B 0,C 180,E1 -22805.509,E2 -22805.509} C_VEL
LIN {X 0,Y 194.715,Z 656.957,A -85,B 0,C 180,E1 -22806.873,E2 -22806.873} C_VEL
LIN {X 0,Y 196.948,Z 643.952,A -85,B 0,C 180,E1 -22807.94,E2 -22807.94} C_VEL
LIN {X 0,Y 198.339,Z 631.138,A -85,B 0,C 180,E1 -22808.623,E2 -22808.623} C_VEL
LIN {X 0,Y 199.254,Z 613.722,A -85,B 0,C 180,E1 -22809.235,E2 -22809.235} C_VEL
LIN {X 0,Y 197.241,Z 579.076,A -85,B 0,C 180,E1 -22811.298,E2 -22811.298} C_VEL
LIN {X 0,Y 195.352,Z 557.825,A -85,B 0,C 180,E1 -22812.787,E2 -22812.787} C_VEL
LIN {X 0,Y 189.751,Z 544.485,A -85,B 0,C 180,E1 -22815,E2 -22815} C_VEL
LIN {X 0,Y 184.955,Z 534.443,A -85,B 0,C 180,E1 -22816.999,E2 -22816.999} C_VEL
LIN {X 0,Y 182.089,Z 528.971,A -85,B 0,C 180,E1 -22818.251,E2 -22818.251} C_VEL
LIN {X 0,Y 179.019,Z 523.364,A -85,B 0,C 180,E1 -22819.656,E2 -22819.656} C_VEL
LIN {X 0,Y 176.132,Z 517.967,A -85,B 0,C 180,E1 -22821.156,E2 -22821.156} C_VEL
LIN {X 0,Y 173.937,Z 511.011,A -85,B 0,C 180,E1 -22825.551,E2 -22825.551} C_VEL
LIN {X 0,Y 171.675,Z 504.186,A -85,B 0,C 180,E1 -22830.577,E2 -22830.577} C_VEL
LIN {X 0,Y 171.459,Z 503.145,A -85,B 0,C 180,E1 -22831.543,E2 -22831.543} C_VEL
LIN {X 0,Y 171.45,Z 503.115,A -85,B 0,C 180,E1 -22835.8,E2 -22835.8} C_VEL
LIN {X 0,Y 171.575,Z 503.062,A -85,B 0,C 180,E1 -22840.871,E2 -22840.871} C_VEL
LIN {X 0,Y 171.573,Z 503.114,A -85,B 0,C 180,E1 -22845.773,E2 -22845.773} C_VEL
LIN {X 0,Y 171.844,Z 503.063,A -85,B 0,C 180,E1 -22850.585,E2 -22850.585} C_VEL
LIN {X 0,Y 171.81,Z 503.056,A -85,B 0,C 180,E1 -22855.307,E2 -22855.307} C_VEL
LIN {X 0,Y 172.33,Z 503.013,A -85,B 0,C 180,E1 -22860,E2 -22860} C_VEL
LIN {X 0,Y 171.812,Z 503.069,A -85,B 0,C 180,E1 -22864.693,E2 -22864.693} C_VEL
LIN {X 0,Y 171.844,Z 503.051,A -85,B 0,C 180,E1 -22869.415,E2 -22869.415} C_VEL
LIN {X 0,Y 171.57,Z 503.1,A -85,B 0,C 180,E1 -22874.228,E2 -22874.228} C_VEL
LIN {X 0,Y 171.539,Z 503.118,A -85,B 0,C 180,E1 -22879.559,E2 -22879.559} C_VEL
LIN {X 0,Y 171.456,Z 503.128,A -85,B 0,C 180,E1 -22885.609,E2 -22885.609} C_VEL
LIN {X 0,Y 171.437,Z 503.054,A -85,B 0,C 180,E1 -22890.586,E2 -22890.586} C_VEL
LIN {X 0,Y 171.372,Z 503.123,A -85,B 0,C 180,E1 -22896.488,E2 -22896.488} C_VEL
LIN {X 0,Y 171.416,Z 503.507,A -85,B 0,C 180,E1 -22897.766,E2 -22897.766} C_VEL
LIN {X 0,Y 171.832,Z 504.872,A -85,B 0,C 180,E1 -22898.321,E2 -22898.321} C_VEL
LIN {X 0,Y 173.301,Z 507.166,A -85,B 0,C 180,E1 -22899.119,E2 -22899.119} C_VEL
LIN {X 0,Y 175.084,Z 508.79,A -85,B 0,C 180,E1 -22899.96,E2 -22899.96} C_VEL
LIN {X 0,Y 177.29,Z 512.193,A -85,B 0,C 180,E1 -22901.045,E2 -22901.045} C_VEL
LIN {X 0,Y 178.726,Z 513.952,A -85,B 0,C 180,E1 -22901.696,E2 -22901.696} C_VEL
LIN {X 0,Y 184.879,Z 522.732,A -85,B 0,C 180,E1 -22904.356,E2 -22904.356} C_VEL
LIN {X 0,Y 191.501,Z 533.066,A -85,B 0,C 180,E1 -22906.947,E2 -22906.947} C_VEL
LIN {X 0,Y 197.832,Z 544.363,A -85,B 0,C 180,E1 -22909.237,E2 -22909.237} C_VEL
LIN {X 0,Y 202.522,Z 553.852,A -85,B 0,C 180,E1 -22910.844,E2 -22910.844} C_VEL
LIN {X 0,Y 201.207,Z 589.184,A -85,B 0,C 180,E1 -22912.204,E2 -22912.204} C_VEL
LIN {X 0,Y 200.046,Z 602.818,A -85,B 0,C 180,E1 -22913.126,E2 -22913.126} C_VEL
LIN {X 0,Y 198.429,Z 614.358,A -85,B 0,C 180,E1 -22914.242,E2 -22914.242} C_VEL
LIN {X 0,Y 196.318,Z 625.5,A -85,B 0,C 180,E1 -22915.674,E2 -22915.674} C_VEL
LIN {X 0,Y 193.356,Z 637.048,A -85,B 0,C 180,E1 -22917.581,E2 -22917.581} C_VEL
LIN {X 0,Y 190.307,Z 647.36,A -85,B 0,C 180,E1 -22919.791,E2 -22919.791} C_VEL
LIN {X 0,Y 187.504,Z 655.766,A -85,B 0,C 180,E1 -22922.062,E2 -22922.062} C_VEL
LIN {X 0,Y 184.704,Z 663.489,A -85,B 0,C 180,E1 -22924.656,E2 -22924.656} C_VEL
LIN {X 0,Y 181.542,Z 671.152,A -85,B 0,C 180,E1 -22927.885,E2 -22927.885} C_VEL
LIN {X 0,Y 178.585,Z 677.95,A -85,B 0,C 180,E1 -22931.65,E2 -22931.65} C_VEL
LIN {X 0,Y 176.393,Z 682.555,A -85,B 0,C 180,E1 -22934.991,E2 -22934.991} C_VEL
LIN {X 0,Y 174.55,Z 686.09,A -85,B 0,C 180,E1 -22938.386,E2 -22938.386} C_VEL
LIN {X 0,Y 173.616,Z 687.911,A -85,B 0,C 180,E1 -22940.682,E2 -22940.682} C_VEL
LIN {X 0,Y 172.78,Z 690.193,A -85,B 0,C 180,E1 -22945.334,E2 -22945.334} C_VEL
LIN {X 0,Y 172.334,Z 691.019,A -85,B 0,C 180,E1 -22950,E2 -22950} C_VEL
LIN {X 0,Y 172.776,Z 690.245,A -85,B 0,C 180,E1 -22954.666,E2 -22954.666} C_VEL
LIN {X 0,Y 173.599,Z 688.017,A -85,B 0,C 180,E1 -22959.319,E2 -22959.319} C_VEL
LIN {X 0,Y 175.153,Z 685.186,A -85,B 0,C 180,E1 -22962.749,E2 -22962.749} C_VEL
LIN {X 0,Y 177.132,Z 681.352,A -85,B 0,C 180,E1 -22966.125,E2 -22966.125} C_VEL
LIN {X 0,Y 179.375,Z 676.265,A -85,B 0,C 180,E1 -22969.571,E2 -22969.571} C_VEL
LIN {X 0,Y 182.048,Z 670.224,A -85,B 0,C 180,E1 -22972.708,E2 -22972.708} C_VEL
LIN {X 0,Y 185.233,Z 662.435,A -85,B 0,C 180,E1 -22975.869,E2 -22975.869} C_VEL
LIN {X 0,Y 188.672,Z 652.753,A -85,B 0,C 180,E1 -22978.962,E2 -22978.962} C_VEL
LIN {X 0,Y 191.589,Z 643.692,A -85,B 0,C 180,E1 -22981.207,E2 -22981.207} C_VEL
LIN {X 0,Y 194.603,Z 633.163,A -85,B 0,C 180,E1 -22983.247,E2 -22983.247} C_VEL
LIN {X 0,Y 197.24,Z 621.617,A -85,B 0,C 180,E1 -22985.008,E2 -22985.008} C_VEL
LIN {X 0,Y 199.368,Z 610.299,A -85,B 0,C 180,E1 -22986.298,E2 -22986.298} C_VEL
LIN {X 0,Y 200.673,Z 598.1,A -85,B 0,C 180,E1 -22987.385,E2 -22987.385} C_VEL
LIN {X 0,Y 201.475,Z 586.337,A -85,B 0,C 180,E1 -22988.076,E2 -22988.076} C_VEL
LIN {X 0,Y 202.562,Z 553.815,A -85,B 0,C 180,E1 -22989.321,E2 -22989.321} C_VEL
LIN {X 0,Y 195.337,Z 539.579,A -85,B 0,C 180,E1 -22991.837,E2 -22991.837} C_VEL
LIN {X 0,Y 188.231,Z 527.789,A -85,B 0,C 180,E1 -22994.499,E2 -22994.499} C_VEL
LIN {X 0,Y 182.882,Z 519.894,A -85,B 0,C 180,E1 -22996.678,E2 -22996.678} C_VEL
LIN {X 0,Y 180.498,Z 516.534,A -85,B 0,C 180,E1 -22997.713,E2 -22997.713} C_VEL
LIN {X 0,Y 177.859,Z 512.752,A -85,B 0,C 180,E1 -22998.921,E2 -22998.921} C_VEL
LIN {X 0,Y 175.546,Z 509.667,A -85,B 0,C 180,E1 -23000.021,E2 -23000.021} C_VEL
LIN {X 0,Y 174.806,Z 508.367,A -85,B 0,C 180,E1 -23000.405,E2 -23000.405} C_VEL
LIN {X 0,Y 172.465,Z 506.115,A -85,B 0,C 180,E1 -23001.54,E2 -23001.54} C_VEL
LIN {X 0,Y 171.452,Z 503.656,A -85,B 0,C 180,E1 -23002.336,E2 -23002.336} C_VEL
LIN {X 0,Y 171.352,Z 503.144,A -85,B 0,C 180,E1 -23003.141,E2 -23003.141} C_VEL
LIN {X 0,Y 171.414,Z 503.065,A -85,B 0,C 180,E1 -23007.791,E2 -23007.791} C_VEL
LIN {X 0,Y 171.444,Z 503.058,A -85,B 0,C 180,E1 -23010.533,E2 -23010.533} C_VEL
LIN {X 0,Y 171.442,Z 503.118,A -85,B 0,C 180,E1 -23015.799,E2 -23015.799} C_VEL
LIN {X 0,Y 171.575,Z 503.113,A -85,B 0,C 180,E1 -23020.871,E2 -23020.871} C_VEL
LIN {X 0,Y 171.588,Z 503.098,A -85,B 0,C 180,E1 -23025.774,E2 -23025.774} C_VEL
LIN {X 0,Y 171.888,Z 503.045,A -85,B 0,C 180,E1 -23030.587,E2 -23030.587} C_VEL
LIN {X 0,Y 171.818,Z 503.065,A -85,B 0,C 180,E1 -23035.307,E2 -23035.307} C_VEL
LIN {X 0,Y 172.33,Z 503.009,A -85,B 0,C 180,E1 -23040,E2 -23040} C_VEL
LIN {X 0,Y 171.81,Z 503.054,A -85,B 0,C 180,E1 -23044.693,E2 -23044.693} C_VEL
LIN {X 0,Y 171.844,Z 503.061,A -85,B 0,C 180,E1 -23049.415,E2 -23049.415} C_VEL
LIN {X 0,Y 171.573,Z 503.114,A -85,B 0,C 180,E1 -23054.227,E2 -23054.227} C_VEL
LIN {X 0,Y 171.539,Z 503.068,A -85,B 0,C 180,E1 -23059.56,E2 -23059.56} C_VEL
LIN {X 0,Y 171.459,Z 503.095,A -85,B 0,C 180,E1 -23065.612,E2 -23065.612} C_VEL
LIN {X 0,Y 171.475,Z 503.359,A -85,B 0,C 180,E1 -23068.621,E2 -23068.621} C_VEL
LIN {X 0,Y 174.015,Z 511.139,A -85,B 0,C 180,E1 -23074.432,E2 -23074.432} C_VEL
LIN {X 0,Y 176.083,Z 517.834,A -85,B 0,C 180,E1 -23078.674,E2 -23078.674} C_VEL
LIN {X 0,Y 179.256,Z 523.694,A -85,B 0,C 180,E1 -23080.329,E2 -23080.329} C_VEL
LIN {X 0,Y 183.915,Z 532.322,A -85,B 0,C 180,E1 -23082.438,E2 -23082.438} C_VEL
LIN {X 0,Y 188.471,Z 541.394,A -85,B 0,C 180,E1 -23084.361,E2 -23084.361} C_VEL
LIN {X 0,Y 195,Z 556.81,A -85,B 0,C 180,E1 -23086.982,E2 -23086.982} C_VEL
LIN {X 0,Y 195.667,Z 559.237,A -85,B 0,C 180,E1 -23087.275,E2 -23087.275} C_VEL
LIN {X 0,Y 197.802,Z 584.938,A -85,B 0,C 180,E1 -23089.028,E2 -23089.028} C_VEL
LIN {X 0,Y 199.398,Z 614.518,A -85,B 0,C 180,E1 -23090.754,E2 -23090.754} C_VEL
LIN {X 0,Y 198.106,Z 635.141,A -85,B 0,C 180,E1 -23091.507,E2 -23091.507} C_VEL
LIN {X 0,Y 196.425,Z 648.32,A -85,B 0,C 180,E1 -23092.323,E2 -23092.323} C_VEL
LIN {X 0,Y 194.021,Z 660.779,A -85,B 0,C 180,E1 -23093.459,E2 -23093.459} C_VEL
LIN {X 0,Y 191.245,Z 672.538,A -85,B 0,C 180,E1 -23094.958,E2 -23094.958} C_VEL
LIN {X 0,Y 187.764,Z 683.879,A -85,B 0,C 180,E1 -23096.811,E2 -23096.811} C_VEL
LIN {X 0,Y 184.172,Z 694.129,A -85,B 0,C 180,E1 -23098.993,E2 -23098.993} C_VEL
LIN {X 0,Y 183.031,Z 697.091,A -85,B 0,C 180,E1 -23099.74,E2 -23099.74} C_VEL
LIN {X 0,Y 180.815,Z 701.351,A -85,B 0,C 180,E1 -23100.829,E2 -23100.829} C_VEL
LIN {X 0,Y 175.616,Z 707.761,A -85,B 0,C 180,E1 -23102.604,E2 -23102.604} C_VEL
LIN {X 0,Y 170.528,Z 713.56,A -85,B 0,C 180,E1 -23104.664,E2 -23104.664} C_VEL
LIN {X 0,Y 168.533,Z 716.859,A -85,B 0,C 180,E1 -23106.175,E2 -23106.175} C_VEL
LIN {X 0,Y 166.281,Z 721.965,A -85,B 0,C 180,E1 -23108.946,E2 -23108.946} C_VEL
LIN {X 0,Y 164.533,Z 727.3,A -85,B 0,C 180,E1 -23112.603,E2 -23112.603} C_VEL
LIN {X 0,Y 163.428,Z 731.492,A -85,B 0,C 180,E1 -23116.319,E2 -23116.319} C_VEL
LIN {X 0,Y 163.08,Z 734.661,A -85,B 0,C 180,E1 -23120.074,E2 -23120.074} C_VEL
LIN {X 0,Y 163.192,Z 736.209,A -85,B 0,C 180,E1 -23122.577,E2 -23122.577} C_VEL
LIN {X 0,Y 163.534,Z 737.35,A -85,B 0,C 180,E1 -23125.069,E2 -23125.069} C_VEL
LIN {X 0,Y 164.627,Z 738.398,A -85,B 0,C 180,E1 -23130,E2 -23130} C_VEL
LIN {X 0,Y 163.549,Z 737.331,A -85,B 0,C 180,E1 -23134.93,E2 -23134.93} C_VEL
LIN {X 0,Y 163.166,Z 735.969,A -85,B 0,C 180,E1 -23137.83,E2 -23137.83} C_VEL
LIN {X 0,Y 163.236,Z 732.583,A -85,B 0,C 180,E1 -23142.431,E2 -23142.431} C_VEL
LIN {X 0,Y 164.113,Z 728.726,A -85,B 0,C 180,E1 -23146.162,E2 -23146.162} C_VEL
LIN {X 0,Y 165.688,Z 723.763,A -85,B 0,C 180,E1 -23149.836,E2 -23149.836} C_VEL
LIN {X 0,Y 168.638,Z 716.435,A -85,B 0,C 180,E1 -23153.973,E2 -23153.973} C_VEL
LIN {X 0,Y 171.857,Z 708.521,A -85,B 0,C 180,E1 -23157.39,E2 -23157.39} C_VEL
LIN {X 0,Y 175.866,Z 698.681,A -85,B 0,C 180,E1 -23160.631,E2 -23160.631} C_VEL
LIN {X 0,Y 179.726,Z 688.573,A -85,B 0,C 180,E1 -23163.192,E2 -23163.192} C_VEL
LIN {X 0,Y 183.632,Z 677.189,A -85,B 0,C 180,E1 -23165.37,E2 -23165.37} C_VEL
LIN {X 0,Y 186.771,Z 666.039,A -85,B 0,C 180,E1 -23167.017,E2 -23167.017} C_VEL
LIN {X 0,Y 189.574,Z 653.679,A -85,B 0,C 180,E1 -23168.386,E2 -23168.386} C_VEL
LIN {X 0,Y 191.671,Z 640.647,A -85,B 0,C 180,E1 -23169.4,E2 -23169.4} C_VEL
LIN {X 0,Y 193.015,Z 627.075,A -85,B 0,C 180,E1 -23170.069,E2 -23170.069} C_VEL
LIN {X 0,Y 193.674,Z 613.979,A -85,B 0,C 180,E1 -23170.535,E2 -23170.535} C_VEL
LIN {X 0,Y 191.952,Z 581.388,A -85,B 0,C 180,E1 -23172.536,E2 -23172.536} C_VEL
LIN {X 0,Y 190.245,Z 560.555,A -85,B 0,C 180,E1 -23174.038,E2 -23174.038} C_VEL
LIN {X 0,Y 183.756,Z 544.995,A -85,B 0,C 180,E1 -23176.805,E2 -23176.805} C_VEL
LIN {X 0,Y 178.338,Z 534.057,A -85,B 0,C 180,E1 -23179.268,E2 -23179.268} C_VEL
LIN {X 0,Y 175.164,Z 528.211,A -85,B 0,C 180,E1 -23180.808,E2 -23180.808} C_VEL
LIN {X 0,Y 171.579,Z 521.863,A -85,B 0,C 180,E1 -23182.663,E2 -23182.663} C_VEL
LIN {X 0,Y 168.235,Z 516.035,A -85,B 0,C 180,E1 -23184.668,E2 -23184.668} C_VEL
LIN {X 0,Y 166.144,Z 509.337,A -85,B 0,C 180,E1 -23189.495,E2 -23189.495} C_VEL
LIN {X 0,Y 164.409,Z 504.042,A -85,B 0,C 180,E1 -23194.114,E2 -23194.114} C_VEL
LIN {X 0,Y 164.482,Z 503.948,A -85,B 0,C 180,E1 -23200.051,E2 -23200.051} C_VEL
LIN {X 0,Y 164.52,Z 503.99,A -85,B 0,C 180,E1 -23205.149,E2 -23205.149} C_VEL
LIN {X 0,Y 164.764,Z 503.94,A -85,B 0,C 180,E1 -23210.176,E2 -23210.176} C_VEL
LIN {X 0,Y 164.827,Z 503.953,A -85,B 0,C 180,E1 -23212.651,E2 -23212.651} C_VEL
LIN {X 0,Y 165.043,Z 503.909,A -85,B 0,C 180,E1 -23217.56,E2 -23217.56} C_VEL
LIN {X 0,Y 165.293,Z 503.889,A -85,B 0,C 180,E1 -23220,E2 -23220} C_VEL
LIN {X 0,Y 164.761,Z 503.949,A -85,B 0,C 180,E1 -23224.894,E2 -23224.894} C_VEL
LIN {X 0,Y 164.828,Z 503.939,A -85,B 0,C 180,E1 -23227.349,E2 -23227.349} C_VEL
LIN {X 0,Y 164.7,Z 503.949,A -85,B 0,C 180,E1 -23231.061,E2 -23231.061} C_VEL
LIN {X 0,Y 164.478,Z 503.977,A -85,B 0,C 180,E1 -23237.404,E2 -23237.404} C_VEL
LIN {X 0,Y 164.47,Z 503.993,A -85,B 0,C 180,E1 -23239.99,E2 -23239.99} C_VEL
LIN {X 0,Y 164.383,Z 503.997,A -85,B 0,C 180,E1 -23246.128,E2 -23246.128} C_VEL
LIN {X 0,Y 164.371,Z 503.933,A -85,B 0,C 180,E1 -23251.227,E2 -23251.227} C_VEL
LIN {X 0,Y 164.386,Z 504.276,A -85,B 0,C 180,E1 -23254.334,E2 -23254.334} C_VEL
LIN {X 0,Y 164.725,Z 505.479,A -85,B 0,C 180,E1 -23254.98,E2 -23254.98} C_VEL
LIN {X 0,Y 166.137,Z 507.917,A -85,B 0,C 180,E1 -23255.903,E2 -23255.903} C_VEL
LIN {X 0,Y 168.295,Z 509.82,A -85,B 0,C 180,E1 -23257.079,E2 -23257.079} C_VEL
LIN {X 0,Y 170.341,Z 513.051,A -85,B 0,C 180,E1 -23258.234,E2 -23258.234} C_VEL
LIN {X 0,Y 172.004,Z 514.834,A -85,B 0,C 180,E1 -23259.076,E2 -23259.076} C_VEL
LIN {X 0,Y 174.594,Z 518.45,A -85,B 0,C 180,E1 -23260.379,E2 -23260.379} C_VEL
LIN {X 0,Y 180.969,Z 527.659,A -85,B 0,C 180,E1 -23263.313,E2 -23263.313} C_VEL
LIN {X 0,Y 187.487,Z 538.055,A -85,B 0,C 180,E1 -23266.013,E2 -23266.013} C_VEL
LIN {X 0,Y 193.677,Z 549.318,A -85,B 0,C 180,E1 -23268.374,E2 -23268.374} C_VEL
LIN {X 0,Y 197.017,Z 556.194,A -85,B 0,C 180,E1 -23269.591,E2 -23269.591} C_VEL
LIN {X 0,Y 195.661,Z 590.619,A -85,B 0,C 180,E1 -23270.965,E2 -23270.965} C_VEL
LIN {X 0,Y 194.452,Z 603.934,A -85,B 0,C 180,E1 -23271.892,E2 -23271.892} C_VEL
LIN {X 0,Y 192.77,Z 615.354,A -85,B 0,C 180,E1 -23273.021,E2 -23273.021} C_VEL
LIN {X 0,Y 190.465,Z 626.891,A -85,B 0,C 180,E1 -23274.544,E2 -23274.544} C_VEL
LIN {X 0,Y 187.46,Z 638.041,A -85,B 0,C 180,E1 -23276.429,E2 -23276.429} C_VEL
LIN {X 0,Y 184.266,Z 648.352,A -85,B 0,C 180,E1 -23278.691,E2 -23278.691} C_VEL
LIN {X 0,Y 181.324,Z 656.757,A -85,B 0,C 180,E1 -23281.022,E2 -23281.022} C_VEL
LIN {X 0,Y 178.377,Z 664.48,A -85,B 0,C 180,E1 -23283.69,E2 -23283.69} C_VEL
LIN {X 0,Y 175.051,Z 672.142,A -85,B 0,C 180,E1 -23287.019,E2 -23287.019} C_VEL
LIN {X 0,Y 171.929,Z 678.94,A -85,B 0,C 180,E1 -23290.913,E2 -23290.913} C_VEL
LIN {X 0,Y 169.615,Z 683.545,A -85,B 0,C 180,E1 -23294.376,E2 -23294.376} C_VEL
LIN {X 0,Y 167.67,Z 687.08,A -85,B 0,C 180,E1 -23297.903,E2 -23297.903} C_VEL
LIN {X 0,Y 166.683,Z 688.9,A -85,B 0,C 180,E1 -23300.291,E2 -23300.291} C_VEL
LIN {X 0,Y 165.776,Z 691.181,A -85,B 0,C 180,E1 -23305.136,E2 -23305.136} C_VEL
LIN {X 0,Y 165.306,Z 692.007,A -85,B 0,C 180,E1 -23310,E2 -23310} C_VEL
LIN {X 0,Y 165.773,Z 691.233,A -85,B 0,C 180,E1 -23314.864,E2 -23314.864} C_VEL
LIN {X 0,Y 166.665,Z 689.005,A -85,B 0,C 180,E1 -23319.71,E2 -23319.71} C_VEL
LIN {X 0,Y 168.305,Z 686.173,A -85,B 0,C 180,E1 -23323.277,E2 -23323.277} C_VEL
LIN {X 0,Y 170.392,Z 682.339,A -85,B 0,C 180,E1 -23326.781,E2 -23326.781} C_VEL
LIN {X 0,Y 172.769,Z 677.251,A -85,B 0,C 180,E1 -23330.352,E2 -23330.352} C_VEL
LIN {X 0,Y 175.586,Z 671.21,A -85,B 0,C 180,E1 -23333.594,E2 -23333.594} C_VEL
LIN {X 0,Y 178.935,Z 663.42,A -85,B 0,C 180,E1 -23336.851,E2 -23336.851} C_VEL
LIN {X 0,Y 182.553,Z 653.738,A -85,B 0,C 180,E1 -23340.031,E2 -23340.031} C_VEL
LIN {X 0,Y 185.614,Z 644.676,A -85,B 0,C 180,E1 -23342.331,E2 -23342.331} C_VEL
LIN {X 0,Y 188.773,Z 634.144,A -85,B 0,C 180,E1 -23344.415,E2 -23344.415} C_VEL
LIN {X 0,Y 191.57,Z 622.443,A -85,B 0,C 180,E1 -23346.234,E2 -23346.234} C_VEL
LIN {X 0,Y 193.801,Z 610.934,A -85,B 0,C 180,E1 -23347.565,E2 -23347.565} C_VEL
LIN {X 0,Y 195.211,Z 598.143,A -85,B 0,C 180,E1 -23348.705,E2 -23348.705} C_VEL
LIN {X 0,Y 196.034,Z 586.224,A -85,B 0,C 180,E1 -23349.393,E2 -23349.393} C_VEL
LIN {X 0,Y 197.038,Z 556.039,A -85,B 0,C 180,E1 -23350.591,E2 -23350.591} C_VEL
LIN {X 0,Y 189.838,Z 542.058,A -85,B 0,C 180,E1 -23353.266,E2 -23353.266} C_VEL
LIN {X 0,Y 182.664,Z 530.181,A -85,B 0,C 180,E1 -23356.167,E2 -23356.167} C_VEL
LIN {X 0,Y 177.046,Z 521.986,A -85,B 0,C 180,E1 -23358.664,E2 -23358.664} C_VEL
LIN {X 0,Y 174.168,Z 517.942,A -85,B 0,C 180,E1 -23360.05,E2 -23360.05} C_VEL
LIN {X 0,Y 171.273,Z 513.94,A -85,B 0,C 180,E1 -23361.531,E2 -23361.531} C_VEL
LIN {X 0,Y 168.903,Z 511.03,A -85,B 0,C 180,E1 -23362.797,E2 -23362.797} C_VEL
LIN {X 0,Y 167.909,Z 509.327,A -85,B 0,C 180,E1 -23363.384,E2 -23363.384} C_VEL
LIN {X 0,Y 165.655,Z 507.326,A -85,B 0,C 180,E1 -23364.636,E2 -23364.636} C_VEL
LIN {X 0,Y 164.442,Z 504.655,A -85,B 0,C 180,E1 -23365.628,E2 -23365.628} C_VEL
LIN {X 0,Y 164.324,Z 504.048,A -85,B 0,C 180,E1 -23366.571,E2 -23366.571} C_VEL
LIN {X 0,Y 164.386,Z 503.931,A -85,B 0,C 180,E1 -23369.133,E2 -23369.133} C_VEL
LIN {X 0,Y 164.403,Z 504.007,A -85,B 0,C 180,E1 -23374.692,E2 -23374.692} C_VEL
LIN {X 0,Y 164.482,Z 503.992,A -85,B 0,C 180,E1 -23380.051,E2 -23380.051} C_VEL
LIN {X 0,Y 164.53,Z 503.97,A -85,B 0,C 180,E1 -23385.15,E2 -23385.15} C_VEL
LIN {X 0,Y 164.802,Z 503.928,A -85,B 0,C 180,E1 -23390.178,E2 -23390.178} C_VEL
LIN {X 0,Y 164.85,Z 503.935,A -85,B 0,C 180,E1 -23392.652,E2 -23392.652} C_VEL
LIN {X 0,Y 165.045,Z 503.895,A -85,B 0,C 180,E1 -23397.559,E2 -23397.559} C_VEL
LIN {X 0,Y 165.293,Z 503.885,A -85,B 0,C 180,E1 -23400,E2 -23400} C_VEL
LIN {X 0,Y 164.759,Z 503.933,A -85,B 0,C 180,E1 -23404.894,E2 -23404.894} C_VEL
LIN {X 0,Y 164.827,Z 503.952,A -85,B 0,C 180,E1 -23407.349,E2 -23407.349} C_VEL
LIN {X 0,Y 164.699,Z 503.942,A -85,B 0,C 180,E1 -23411.061,E2 -23411.061} C_VEL
LIN {X 0,Y 164.478,Z 503.952,A -85,B 0,C 180,E1 -23417.404,E2 -23417.404} C_VEL
LIN {X 0,Y 164.47,Z 503.95,A -85,B 0,C 180,E1 -23419.99,E2 -23419.99} C_VEL
LIN {X 0,Y 164.415,Z 504.109,A -85,B 0,C 180,E1 -23425.885,E2 -23425.885} C_VEL
LIN {X 0,Y 166.608,Z 510.86,A -85,B 0,C 180,E1 -23431.542,E2 -23431.542} C_VEL
LIN {X 0,Y 168.273,Z 516.104,A -85,B 0,C 180,E1 -23435.232,E2 -23435.232} C_VEL
LIN {X 0,Y 172.01,Z 522.475,A -85,B 0,C 180,E1 -23437.421,E2 -23437.421} C_VEL
LIN {X 0,Y 176.896,Z 531.334,A -85,B 0,C 180,E1 -23439.918,E2 -23439.918} C_VEL
LIN {X 0,Y 180.165,Z 537.619,A -85,B 0,C 180,E1 -23441.47,E2 -23441.47} C_VEL
LIN {X 0,Y 184.142,Z 545.756,A -85,B 0,C 180,E1 -23443.254,E2 -23443.254} C_VEL
LIN {X 0,Y 190.217,Z 560.412,A -85,B 0,C 180,E1 -23445.851,E2 -23445.851} C_VEL
LIN {X 0,Y 190.8,Z 564.853,A -85,B 0,C 180,E1 -23446.239,E2 -23446.239} C_VEL
LIN {X 0,Y 192.718,Z 591.99,A -85,B 0,C 180,E1 -23448.089,E2 -23448.089} C_VEL
LIN {X 0,Y 193.813,Z 615.978,A -85,B 0,C 180,E1 -23449.508,E2 -23449.508} C_VEL
LIN {X 0,Y 192.491,Z 635.112,A -85,B 0,C 180,E1 -23450.236,E2 -23450.236} C_VEL
LIN {X 0,Y 190.729,Z 648.08,A -85,B 0,C 180,E1 -23451.077,E2 -23451.077} C_VEL
LIN {X 0,Y 188.12,Z 660.785,A -85,B 0,C 180,E1 -23452.285,E2 -23452.285} C_VEL
LIN {X 0,Y 185.008,Z 673.134,A -85,B 0,C 180,E1 -23453.929,E2 -23453.929} C_VEL
LIN {X 0,Y 181.416,Z 684.146,A -85,B 0,C 180,E1 -23455.826,E2 -23455.826} C_VEL
LIN {X 0,Y 177.316,Z 695.105,A -85,B 0,C 180,E1 -23458.321,E2 -23458.321} C_VEL
LIN {X 0,Y 173.761,Z 704.059,A -85,B 0,C 180,E1 -23460.965,E2 -23460.965} C_VEL
LIN {X 0,Y 170.155,Z 712.843,A -85,B 0,C 180,E1 -23464.299,E2 -23464.299} C_VEL
LIN {X 0,Y 168.533,Z 716.859,A -85,B 0,C 180,E1 -23466.175,E2 -23466.175} C_VEL
LIN {X 0,Y 166.629,Z 719.982,A -85,B 0,C 180,E1 -23467.777,E2 -23467.777} C_VEL
LIN {X 0,Y 162.027,Z 724.398,A -85,B 0,C 180,E1 -23470.435,E2 -23470.435} C_VEL
LIN {X 0,Y 157.808,Z 728.104,A -85,B 0,C 180,E1 -23473.357,E2 -23473.357} C_VEL
LIN {X 0,Y 156.547,Z 730.104,A -85,B 0,C 180,E1 -23475.317,E2 -23475.317} C_VEL
LIN {X 0,Y 156.008,Z 733.651,A -85,B 0,C 180,E1 -23479.619,E2 -23479.619} C_VEL
LIN {X 0,Y 156.135,Z 735.208,A -85,B 0,C 180,E1 -23482.239,E2 -23482.239} C_VEL
LIN {X 0,Y 156.431,Z 736.348,A -85,B 0,C 180,E1 -23484.845,E2 -23484.845} C_VEL
LIN {X 0,Y 156.87,Z 737.076,A -85,B 0,C 180,E1 -23487.432,E2 -23487.432} C_VEL
LIN {X 0,Y 157.544,Z 737.402,A -85,B 0,C 180,E1 -23490,E2 -23490} C_VEL
LIN {X 0,Y 156.882,Z 737.064,A -85,B 0,C 180,E1 -23492.568,E2 -23492.568} C_VEL
LIN {X 0,Y 156.443,Z 736.328,A -85,B 0,C 180,E1 -23495.155,E2 -23495.155} C_VEL
LIN {X 0,Y 156.097,Z 735.107,A -85,B 0,C 180,E1 -23497.899,E2 -23497.899} C_VEL
LIN {X 0,Y 156.097,Z 732.634,A -85,B 0,C 180,E1 -23501.689,E2 -23501.689} C_VEL
LIN {X 0,Y 156.798,Z 729.11,A -85,B 0,C 180,E1 -23505.6,E2 -23505.6} C_VEL
LIN {X 0,Y 158.307,Z 724.533,A -85,B 0,C 180,E1 -23509.448,E2 -23509.448} C_VEL
LIN {X 0,Y 160.883,Z 718.325,A -85,B 0,C 180,E1 -23513.456,E2 -23513.456} C_VEL
LIN {X 0,Y 164.323,Z 710.323,A -85,B 0,C 180,E1 -23517.372,E2 -23517.372} C_VEL
LIN {X 0,Y 168.312,Z 701.207,A -85,B 0,C 180,E1 -23520.764,E2 -23520.764} C_VEL
LIN {X 0,Y 172.089,Z 691.876,A -85,B 0,C 180,E1 -23523.457,E2 -23523.457} C_VEL
LIN {X 0,Y 176.029,Z 681.561,A -85,B 0,C 180,E1 -23525.725,E2 -23525.725} C_VEL
LIN {X 0,Y 179.736,Z 670.14,A -85,B 0,C 180,E1 -23527.658,E2 -23527.658} C_VEL
LIN {X 0,Y 182.801,Z 658.279,A -85,B 0,C 180,E1 -23529.194,E2 -23529.194} C_VEL
LIN {X 0,Y 185.381,Z 645.483,A -85,B 0,C 180,E1 -23530.369,E2 -23530.369} C_VEL
LIN {X 0,Y 187.122,Z 632.27,A -85,B 0,C 180,E1 -23531.198,E2 -23531.198} C_VEL
LIN {X 0,Y 188.222,Z 614.914,A -85,B 0,C 180,E1 -23531.872,E2 -23531.872} C_VEL
LIN {X 0,Y 186.675,Z 582.593,A -85,B 0,C 180,E1 -23533.925,E2 -23533.925} C_VEL
LIN {X 0,Y 185.143,Z 563.163,A -85,B 0,C 180,E1 -23535.391,E2 -23535.391} C_VEL
LIN {X 0,Y 179.335,Z 549.058,A -85,B 0,C 180,E1 -23538.042,E2 -23538.042} C_VEL
LIN {X 0,Y 174.686,Z 539.265,A -85,B 0,C 180,E1 -23540.306,E2 -23540.306} C_VEL
LIN {X 0,Y 171.256,Z 532.807,A -85,B 0,C 180,E1 -23542.079,E2 -23542.079} C_VEL
LIN {X 0,Y 168.133,Z 527.119,A -85,B 0,C 180,E1 -23543.807,E2 -23543.807} C_VEL
LIN {X 0,Y 164.142,Z 520.482,A -85,B 0,C 180,E1 -23546.178,E2 -23546.178} C_VEL
LIN {X 0,Y 160.398,Z 514.065,A -85,B 0,C 180,E1 -23548.83,E2 -23548.83} C_VEL
LIN {X 0,Y 158.503,Z 508.298,A -85,B 0,C 180,E1 -23553.679,E2 -23553.679} C_VEL
LIN {X 0,Y 157.331,Z 504.925,A -85,B 0,C 180,E1 -23557.166,E2 -23557.166} C_VEL
LIN {X 0,Y 157.405,Z 504.827,A -85,B 0,C 180,E1 -23561.787,E2 -23561.787} C_VEL
LIN {X 0,Y 157.526,Z 504.846,A -85,B 0,C 180,E1 -23567.11,E2 -23567.11} C_VEL
LIN {X 0,Y 157.783,Z 504.832,A -85,B 0,C 180,E1 -23572.321,E2 -23572.321} C_VEL
LIN {X 0,Y 158.255,Z 504.764,A -85,B 0,C 180,E1 -23580,E2 -23580} C_VEL
LIN {X 0,Y 157.764,Z 504.814,A -85,B 0,C 180,E1 -23587.68,E2 -23587.68} C_VEL
LIN {X 0,Y 157.634,Z 504.83,A -85,B 0,C 180,E1 -23591.236,E2 -23591.236} C_VEL
LIN {X 0,Y 157.437,Z 504.849,A -85,B 0,C 180,E1 -23595.536,E2 -23595.536} C_VEL
LIN {X 0,Y 157.365,Z 504.866,A -85,B 0,C 180,E1 -23600.934,E2 -23600.934} C_VEL
LIN {X 0,Y 157.307,Z 504.86,A -85,B 0,C 180,E1 -23606.681,E2 -23606.681} C_VEL
LIN {X 0,Y 157.344,Z 505.143,A -85,B 0,C 180,E1 -23610.258,E2 -23610.258} C_VEL
LIN {X 0,Y 157.671,Z 506.22,A -85,B 0,C 180,E1 -23611.025,E2 -23611.025} C_VEL
LIN {X 0,Y 159.043,Z 508.703,A -85,B 0,C 180,E1 -23612.117,E2 -23612.117} C_VEL
LIN {X 0,Y 161.51,Z 510.675,A -85,B 0,C 180,E1 -23613.698,E2 -23613.698} C_VEL
LIN {X 0,Y 163.348,Z 513.837,A -85,B 0,C 180,E1 -23614.934,E2 -23614.934} C_VEL
LIN {X 0,Y 165.477,Z 516.05,A -85,B 0,C 180,E1 -23616.179,E2 -23616.179} C_VEL
LIN {X 0,Y 167.996,Z 519.558,A -85,B 0,C 180,E1 -23617.627,E2 -23617.627} C_VEL
LIN {X 0,Y 169.434,Z 521.505,A -85,B 0,C 180,E1 -23618.41,E2 -23618.41} C_VEL
LIN {X 0,Y 172.997,Z 526.586,A -85,B 0,C 180,E1 -23620.255,E2 -23620.255} C_VEL
LIN {X 0,Y 177.469,Z 533.163,A -85,B 0,C 180,E1 -23622.387,E2 -23622.387} C_VEL
LIN {X 0,Y 183.547,Z 543.06,A -85,B 0,C 180,E1 -23625.046,E2 -23625.046} C_VEL
LIN {X 0,Y 189.574,Z 554.364,A -85,B 0,C 180,E1 -23627.481,E2 -23627.481} C_VEL
LIN {X 0,Y 191.634,Z 558.711,A -85,B 0,C 180,E1 -23628.28,E2 -23628.28} C_VEL
LIN {X 0,Y 190.24,Z 591.596,A -85,B 0,C 180,E1 -23629.626,E2 -23629.626} C_VEL
LIN {X 0,Y 188.955,Z 605.053,A -85,B 0,C 180,E1 -23630.586,E2 -23630.586} C_VEL
LIN {X 0,Y 187.201,Z 616.35,A -85,B 0,C 180,E1 -23631.726,E2 -23631.726} C_VEL
LIN {X 0,Y 184.878,Z 627.494,A -85,B 0,C 180,E1 -23633.217,E2 -23633.217} C_VEL
LIN {X 0,Y 181.646,Z 639.033,A -85,B 0,C 180,E1 -23635.203,E2 -23635.203} C_VEL
LIN {X 0,Y 178.298,Z 649.344,A -85,B 0,C 180,E1 -23637.517,E2 -23637.517} C_VEL
LIN {X 0,Y 175.209,Z 657.749,A -85,B 0,C 180,E1 -23639.908,E2 -23639.908} C_VEL
LIN {X 0,Y 172.105,Z 665.47,A -85,B 0,C 180,E1 -23642.652,E2 -23642.652} C_VEL
LIN {X 0,Y 168.603,Z 673.132,A -85,B 0,C 180,E1 -23646.086,E2 -23646.086} C_VEL
LIN {X 0,Y 165.303,Z 679.929,A -85,B 0,C 180,E1 -23650.116,E2 -23650.116} C_VEL
LIN {X 0,Y 162.857,Z 684.534,A -85,B 0,C 180,E1 -23653.71,E2 -23653.71} C_VEL
LIN {X 0,Y 160.803,Z 688.069,A -85,B 0,C 180,E1 -23657.378,E2 -23657.378} C_VEL
LIN {X 0,Y 159.757,Z 689.889,A -85,B 0,C 180,E1 -23659.865,E2 -23659.865} C_VEL
LIN {X 0,Y 158.775,Z 692.17,A -85,B 0,C 180,E1 -23664.921,E2 -23664.921} C_VEL
LIN {X 0,Y 158.278,Z 692.995,A -85,B 0,C 180,E1 -23670,E2 -23670} C_VEL
LIN {X 0,Y 158.772,Z 692.22,A -85,B 0,C 180,E1 -23675.079,E2 -23675.079} C_VEL
LIN {X 0,Y 159.74,Z 689.993,A -85,B 0,C 180,E1 -23680.136,E2 -23680.136} C_VEL
LIN {X 0,Y 161.473,Z 687.16,A -85,B 0,C 180,E1 -23683.85,E2 -23683.85} C_VEL
LIN {X 0,Y 163.676,Z 683.326,A -85,B 0,C 180,E1 -23687.491,E2 -23687.491} C_VEL
LIN {X 0,Y 166.197,Z 678.238,A -85,B 0,C 180,E1 -23691.194,E2 -23691.194} C_VEL
LIN {X 0,Y 169.169,Z 672.197,A -85,B 0,C 180,E1 -23694.547,E2 -23694.547} C_VEL
LIN {X 0,Y 172.694,Z 664.406,A -85,B 0,C 180,E1 -23697.904,E2 -23697.904} C_VEL
LIN {X 0,Y 176.502,Z 654.723,A -85,B 0,C 180,E1 -23701.173,E2 -23701.173} C_VEL
LIN {X 0,Y 179.715,Z 645.66,A -85,B 0,C 180,E1 -23703.529,E2 -23703.529} C_VEL
LIN {X 0,Y 183.018,Z 635.127,A -85,B 0,C 180,E1 -23705.659,E2 -23705.659} C_VEL
LIN {X 0,Y 185.902,Z 623.582,A -85,B 0,C 180,E1 -23707.495,E2 -23707.495} C_VEL
LIN {X 0,Y 188.224,Z 612.26,A -85,B 0,C 180,E1 -23708.832,E2 -23708.832} C_VEL
LIN {X 0,Y 189.768,Z 599.213,A -85,B 0,C 180,E1 -23710.025,E2 -23710.025} C_VEL
LIN {X 0,Y 190.649,Z 587.193,A -85,B 0,C 180,E1 -23710.735,E2 -23710.735} C_VEL
LIN {X 0,Y 191.672,Z 558.644,A -85,B 0,C 180,E1 -23711.898,E2 -23711.898} C_VEL
LIN {X 0,Y 185.519,Z 546.459,A -85,B 0,C 180,E1 -23714.341,E2 -23714.341} C_VEL
LIN {X 0,Y 178.944,Z 535.37,A -85,B 0,C 180,E1 -23717.16,E2 -23717.16} C_VEL
LIN {X 0,Y 173.265,Z 526.9,A -85,B 0,C 180,E1 -23719.841,E2 -23719.841} C_VEL
LIN {X 0,Y 170.755,Z 523.354,A -85,B 0,C 180,E1 -23721.123,E2 -23721.123} C_VEL
LIN {X 0,Y 168.067,Z 519.586,A -85,B 0,C 180,E1 -23722.58,E2 -23722.58} C_VEL
LIN {X 0,Y 165.547,Z 516.146,A -85,B 0,C 180,E1 -23724.032,E2 -23724.032} C_VEL
LIN {X 0,Y 164.43,Z 514.897,A -85,B 0,C 180,E1 -23724.686,E2 -23724.686} C_VEL
LIN {X 0,Y 162.287,Z 512.262,A -85,B 0,C 180,E1 -23726.019,E2 -23726.019} C_VEL
LIN {X 0,Y 161.176,Z 510.387,A -85,B 0,C 180,E1 -23726.785,E2 -23726.785} C_VEL
LIN {X 0,Y 158.497,Z 507.928,A -85,B 0,C 180,E1 -23728.568,E2 -23728.568} C_VEL
LIN {X 0,Y 157.425,Z 505.501,A -85,B 0,C 180,E1 -23729.667,E2 -23729.667} C_VEL
LIN {X 0,Y 157.295,Z 504.916,A -85,B 0,C 180,E1 -23730.562,E2 -23730.562} C_VEL
LIN {X 0,Y 157.311,Z 504.862,A -85,B 0,C 180,E1 -23733.464,E2 -23733.464} C_VEL
LIN {X 0,Y 157.389,Z 504.869,A -85,B 0,C 180,E1 -23739.669,E2 -23739.669} C_VEL
LIN {X 0,Y 157.456,Z 504.847,A -85,B 0,C 180,E1 -23744.466,E2 -23744.466} C_VEL
LIN {X 0,Y 157.725,Z 504.811,A -85,B 0,C 180,E1 -23749.733,E2 -23749.733} C_VEL
LIN {X 0,Y 157.807,Z 504.808,A -85,B 0,C 180,E1 -23752.322,E2 -23752.322} C_VEL
LIN {X 0,Y 158.255,Z 504.76,A -85,B 0,C 180,E1 -23760,E2 -23760} C_VEL
LIN {X 0,Y 157.783,Z 504.831,A -85,B 0,C 180,E1 -23767.679,E2 -23767.679} C_VEL
LIN {X 0,Y 157.526,Z 504.847,A -85,B 0,C 180,E1 -23772.89,E2 -23772.89} C_VEL
LIN {X 0,Y 157.405,Z 504.827,A -85,B 0,C 180,E1 -23778.213,E2 -23778.213} C_VEL
LIN {X 0,Y 157.342,Z 505.073,A -85,B 0,C 180,E1 -23782.92,E2 -23782.92} C_VEL
LIN {X 0,Y 159.162,Z 510.312,A -85,B 0,C 180,E1 -23787.981,E2 -23787.981} C_VEL
LIN {X 0,Y 160.51,Z 514.323,A -85,B 0,C 180,E1 -23791.146,E2 -23791.146} C_VEL
LIN {X 0,Y 165.641,Z 522.846,A -85,B 0,C 180,E1 -23794.575,E2 -23794.575} C_VEL
LIN {X 0,Y 169.528,Z 529.523,A -85,B 0,C 180,E1 -23796.829,E2 -23796.829} C_VEL
LIN {X 0,Y 173.409,Z 536.82,A -85,B 0,C 180,E1 -23798.917,E2 -23798.917} C_VEL
LIN {X 0,Y 176.192,Z 542.294,A -85,B 0,C 180,E1 -23800.32,E2 -23800.32} C_VEL
LIN {X 0,Y 180.151,Z 550.753,A -85,B 0,C 180,E1 -23802.219,E2 -23802.219} C_VEL
LIN {X 0,Y 185.347,Z 563.553,A -85,B 0,C 180,E1 -23804.589,E2 -23804.589} C_VEL
LIN {X 0,Y 186.949,Z 584.708,A -85,B 0,C 180,E1 -23806.164,E2 -23806.164} C_VEL
LIN {X 0,Y 188.409,Z 615.476,A -85,B 0,C 180,E1 -23808.113,E2 -23808.113} C_VEL
LIN {X 0,Y 187.06,Z 634.13,A -85,B 0,C 180,E1 -23808.838,E2 -23808.838} C_VEL
LIN {X 0,Y 185.247,Z 647.183,A -85,B 0,C 180,E1 -23809.706,E2 -23809.706} C_VEL
LIN {X 0,Y 182.568,Z 659.795,A -85,B 0,C 180,E1 -23810.924,E2 -23810.924} C_VEL
LIN {X 0,Y 179.299,Z 672.137,A -85,B 0,C 180,E1 -23812.588,E2 -23812.588} C_VEL
LIN {X 0,Y 175.549,Z 683.145,A -85,B 0,C 180,E1 -23814.515,E2 -23814.515} C_VEL
LIN {X 0,Y 171.319,Z 694.11,A -85,B 0,C 180,E1 -23817.075,E2 -23817.075} C_VEL
LIN {X 0,Y 167.565,Z 703.06,A -85,B 0,C 180,E1 -23819.782,E2 -23819.782} C_VEL
LIN {X 0,Y 164.328,Z 710.491,A -85,B 0,C 180,E1 -23822.629,E2 -23822.629} C_VEL
LIN {X 0,Y 160.954,Z 718.345,A -85,B 0,C 180,E1 -23826.485,E2 -23826.485} C_VEL
LIN {X 0,Y 158.886,Z 722.853,A -85,B 0,C 180,E1 -23829.277,E2 -23829.277} C_VEL
LIN {X 0,Y 157.21,Z 727.8,A -85,B 0,C 180,E1 -23833.108,E2 -23833.108} C_VEL
LIN {X 0,Y 156.547,Z 730.104,A -85,B 0,C 180,E1 -23835.317,E2 -23835.317} C_VEL
LIN {X 0,Y 155.505,Z 731.906,A -85,B 0,C 180,E1 -23837.349,E2 -23837.349} C_VEL
LIN {X 0,Y 152.476,Z 733.999,A -85,B 0,C 180,E1 -23840.776,E2 -23840.776} C_VEL
LIN {X 0,Y 150.276,Z 735.15,A -85,B 0,C 180,E1 -23843.653,E2 -23843.653} C_VEL
LIN {X 0,Y 149.585,Z 735.769,A -85,B 0,C 180,E1 -23845.899,E2 -23845.899} C_VEL
LIN {X 0,Y 149.647,Z 735.902,A -85,B 0,C 180,E1 -23846.654,E2 -23846.654} C_VEL
LIN {X 0,Y 150.461,Z 736.406,A -85,B 0,C 180,E1 -23850,E2 -23850} C_VEL
LIN {X 0,Y 149.798,Z 736.067,A -85,B 0,C 180,E1 -23852.689,E2 -23852.689} C_VEL
LIN {X 0,Y 149.346,Z 735.325,A -85,B 0,C 180,E1 -23855.4,E2 -23855.4} C_VEL
LIN {X 0,Y 149.04,Z 734.171,A -85,B 0,C 180,E1 -23858.132,E2 -23858.132} C_VEL
LIN {X 0,Y 149.081,Z 731.625,A -85,B 0,C 180,E1 -23862.247,E2 -23862.247} C_VEL
LIN {X 0,Y 149.898,Z 728.1,A -85,B 0,C 180,E1 -23866.338,E2 -23866.338} C_VEL
LIN {X 0,Y 151.55,Z 723.522,A -85,B 0,C 180,E1 -23870.353,E2 -23870.353} C_VEL
LIN {X 0,Y 154.63,Z 716.723,A -85,B 0,C 180,E1 -23874.86,E2 -23874.86} C_VEL
LIN {X 0,Y 158.011,Z 709.316,A -85,B 0,C 180,E1 -23878.563,E2 -23878.563} C_VEL
LIN {X 0,Y 162.226,Z 700.202,A -85,B 0,C 180,E1 -23882.052,E2 -23882.052} C_VEL
LIN {X 0,Y 166.197,Z 690.872,A -85,B 0,C 180,E1 -23884.81,E2 -23884.81} C_VEL
LIN {X 0,Y 170.311,Z 680.558,A -85,B 0,C 180,E1 -23887.121,E2 -23887.121} C_VEL
LIN {X 0,Y 174.136,Z 669.13,A -85,B 0,C 180,E1 -23889.094,E2 -23889.094} C_VEL
LIN {X 0,Y 177.357,Z 657.275,A -85,B 0,C 180,E1 -23890.643,E2 -23890.643} C_VEL
LIN {X 0,Y 179.944,Z 644.675,A -85,B 0,C 180,E1 -23891.832,E2 -23891.832} C_VEL
LIN {X 0,Y 181.835,Z 631.251,A -85,B 0,C 180,E1 -23892.673,E2 -23892.673} C_VEL
LIN {X 0,Y 182.892,Z 615.836,A -85,B 0,C 180,E1 -23893.284,E2 -23893.284} C_VEL
LIN {X 0,Y 181.492,Z 583.378,A -85,B 0,C 180,E1 -23895.423,E2 -23895.423} C_VEL
LIN {X 0,Y 180.266,Z 566.197,A -85,B 0,C 180,E1 -23896.759,E2 -23896.759} C_VEL
LIN {X 0,Y 175.234,Z 553.518,A -85,B 0,C 180,E1 -23899.232,E2 -23899.232} C_VEL
LIN {X 0,Y 170.628,Z 543.578,A -85,B 0,C 180,E1 -23901.635,E2 -23901.635} C_VEL
LIN {X 0,Y 167.509,Z 537.546,A -85,B 0,C 180,E1 -23903.367,E2 -23903.367} C_VEL
LIN {X 0,Y 164.617,Z 532.11,A -85,B 0,C 180,E1 -23905.086,E2 -23905.086} C_VEL
LIN {X 0,Y 161.052,Z 525.946,A -85,B 0,C 180,E1 -23907.358,E2 -23907.358} C_VEL
LIN {X 0,Y 156.814,Z 518.948,A -85,B 0,C 180,E1 -23910.37,E2 -23910.37} C_VEL
LIN {X 0,Y 152.523,Z 512.034,A -85,B 0,C 180,E1 -23914.04,E2 -23914.04} C_VEL
LIN {X 0,Y 150.538,Z 506.647,A -85,B 0,C 180,E1 -23919.572,E2 -23919.572} C_VEL
LIN {X 0,Y 150.356,Z 505.784,A -85,B 0,C 180,E1 -23920.901,E2 -23920.901} C_VEL
LIN {X 0,Y 150.433,Z 505.736,A -85,B 0,C 180,E1 -23926.491,E2 -23926.491} C_VEL
LIN {X 0,Y 150.608,Z 505.698,A -85,B 0,C 180,E1 -23929.242,E2 -23929.242} C_VEL
LIN {X 0,Y 150.716,Z 505.71,A -85,B 0,C 180,E1 -23931.958,E2 -23931.958} C_VEL
LIN {X 0,Y 151.215,Z 505.64,A -85,B 0,C 180,E1 -23940,E2 -23940} C_VEL
LIN {X 0,Y 150.702,Z 505.689,A -85,B 0,C 180,E1 -23948.043,E2 -23948.043} C_VEL
LIN {X 0,Y 150.574,Z 505.711,A -85,B 0,C 180,E1 -23951.437,E2 -23951.437} C_VEL
LIN {X 0,Y 150.348,Z 505.731,A -85,B 0,C 180,E1 -23956.288,E2 -23956.288} C_VEL
LIN {X 0,Y 150.347,Z 505.741,A -85,B 0,C 180,E1 -23960.791,E2 -23960.791} C_VEL
LIN {X 0,Y 150.273,Z 506.027,A -85,B 0,C 180,E1 -23965.155,E2 -23965.155} C_VEL
LIN {X 0,Y 150.596,Z 507.188,A -85,B 0,C 180,E1 -23966.084,E2 -23966.084} C_VEL
LIN {X 0,Y 152.194,Z 509.841,A -85,B 0,C 180,E1 -23967.653,E2 -23967.653} C_VEL
LIN {X 0,Y 154.88,Z 511.812,A -85,B 0,C 180,E1 -23969.757,E2 -23969.757} C_VEL
LIN {X 0,Y 156.566,Z 514.794,A -85,B 0,C 180,E1 -23971.13,E2 -23971.13} C_VEL
LIN {X 0,Y 158.97,Z 517.147,A -85,B 0,C 180,E1 -23972.791,E2 -23972.791} C_VEL
LIN {X 0,Y 161.314,Z 520.558,A -85,B 0,C 180,E1 -23974.381,E2 -23974.381} C_VEL
LIN {X 0,Y 162.776,Z 522.226,A -85,B 0,C 180,E1 -23975.283,E2 -23975.283} C_VEL
LIN {X 0,Y 166.633,Z 527.656,A -85,B 0,C 180,E1 -23977.57,E2 -23977.57} C_VEL
LIN {X 0,Y 169.776,Z 532.185,A -85,B 0,C 180,E1 -23979.281,E2 -23979.281} C_VEL
LIN {X 0,Y 175.651,Z 541.128,A -85,B 0,C 180,E1 -23982.196,E2 -23982.196} C_VEL
LIN {X 0,Y 182.027,Z 552.38,A -85,B 0,C 180,E1 -23985.069,E2 -23985.069} C_VEL
LIN {X 0,Y 186.326,Z 561.183,A -85,B 0,C 180,E1 -23986.884,E2 -23986.884} C_VEL
LIN {X 0,Y 184.925,Z 592.603,A -85,B 0,C 180,E1 -23988.211,E2 -23988.211} C_VEL
LIN {X 0,Y 183.559,Z 606.183,A -85,B 0,C 180,E1 -23989.204,E2 -23989.204} C_VEL
LIN {X 0,Y 181.734,Z 617.346,A -85,B 0,C 180,E1 -23990.353,E2 -23990.353} C_VEL
LIN {X 0,Y 179.299,Z 628.487,A -85,B 0,C 180,E1 -23991.873,E2 -23991.873} C_VEL
LIN {X 0,Y 175.922,Z 640.026,A -85,B 0,C 180,E1 -23993.897,E2 -23993.897} C_VEL
LIN {X 0,Y 172.41,Z 650.335,A -85,B 0,C 180,E1 -23996.263,E2 -23996.263} C_VEL
LIN {X 0,Y 169.164,Z 658.74,A -85,B 0,C 180,E1 -23998.714,E2 -23998.714} C_VEL
LIN {X 0,Y 165.894,Z 666.461,A -85,B 0,C 180,E1 -24001.537,E2 -24001.537} C_VEL
LIN {X 0,Y 162.203,Z 674.122,A -85,B 0,C 180,E1 -24005.08,E2 -24005.08} C_VEL
LIN {X 0,Y 158.712,Z 680.919,A -85,B 0,C 180,E1 -24009.253,E2 -24009.253} C_VEL
LIN {X 0,Y 156.124,Z 685.523,A -85,B 0,C 180,E1 -24012.987,E2 -24012.987} C_VEL
LIN {X 0,Y 153.951,Z 689.058,A -85,B 0,C 180,E1 -24016.806,E2 -24016.806} C_VEL
LIN {X 0,Y 152.841,Z 690.879,A -85,B 0,C 180,E1 -24019.402,E2 -24019.402} C_VEL
LIN {X 0,Y 151.776,Z 693.158,A -85,B 0,C 180,E1 -24024.686,E2 -24024.686} C_VEL
LIN {X 0,Y 151.25,Z 693.984,A -85,B 0,C 180,E1 -24030,E2 -24030} C_VEL
LIN {X 0,Y 151.773,Z 693.208,A -85,B 0,C 180,E1 -24035.314,E2 -24035.314} C_VEL
LIN {X 0,Y 152.824,Z 690.981,A -85,B 0,C 180,E1 -24040.6,E2 -24040.6} C_VEL
LIN {X 0,Y 154.659,Z 688.147,A -85,B 0,C 180,E1 -24044.473,E2 -24044.473} C_VEL
LIN {X 0,Y 156.987,Z 684.313,A -85,B 0,C 180,E1 -24048.262,E2 -24048.262} C_VEL
LIN {X 0,Y 159.665,Z 679.224,A -85,B 0,C 180,E1 -24052.106,E2 -24052.106} C_VEL
LIN {X 0,Y 162.802,Z 673.183,A -85,B 0,C 180,E1 -24055.574,E2 -24055.574} C_VEL
LIN {X 0,Y 166.515,Z 665.392,A -85,B 0,C 180,E1 -24059.036,E2 -24059.036} C_VEL
LIN {X 0,Y 170.527,Z 655.709,A -85,B 0,C 180,E1 -24062.396,E2 -24062.396} C_VEL
LIN {X 0,Y 173.9,Z 646.645,A -85,B 0,C 180,E1 -24064.808,E2 -24064.808} C_VEL
LIN {X 0,Y 177.347,Z 636.113,A -85,B 0,C 180,E1 -24066.984,E2 -24066.984} C_VEL
LIN {X 0,Y 180.378,Z 624.564,A -85,B 0,C 180,E1 -24068.853,E2 -24068.853} C_VEL
LIN {X 0,Y 182.801,Z 613.241,A -85,B 0,C 180,E1 -24070.214,E2 -24070.214} C_VEL
LIN {X 0,Y 184.432,Z 600.394,A -85,B 0,C 180,E1 -24071.411,E2 -24071.411} C_VEL
LIN {X 0,Y 185.375,Z 587.894,A -85,B 0,C 180,E1 -24072.171,E2 -24072.171} C_VEL
LIN {X 0,Y 186.392,Z 561.179,A -85,B 0,C 180,E1 -24073.29,E2 -24073.29} C_VEL
LIN {X 0,Y 180.899,Z 550.198,A -85,B 0,C 180,E1 -24075.628,E2 -24075.628} C_VEL
LIN {X 0,Y 175.066,Z 540.246,A -85,B 0,C 180,E1 -24078.295,E2 -24078.295} C_VEL
LIN {X 0,Y 170.116,Z 532.612,A -85,B 0,C 180,E1 -24080.778,E2 -24080.778} C_VEL
LIN {X 0,Y 165.151,Z 525.443,A -85,B 0,C 180,E1 -24083.541,E2 -24083.541} C_VEL
LIN {X 0,Y 161.885,Z 521.108,A -85,B 0,C 180,E1 -24085.535,E2 -24085.535} C_VEL
LIN {X 0,Y 159.452,Z 517.955,A -85,B 0,C 180,E1 -24087.142,E2 -24087.142} C_VEL
LIN {X 0,Y 158.464,Z 516.51,A -85,B 0,C 180,E1 -24087.845,E2 -24087.845} C_VEL
LIN {X 0,Y 155.885,Z 513.751,A -85,B 0,C 180,E1 -24089.701,E2 -24089.701} C_VEL
LIN {X 0,Y 154.635,Z 511.482,A -85,B 0,C 180,E1 -24090.753,E2 -24090.753} C_VEL
LIN {X 0,Y 152.064,Z 509.69,A -85,B 0,C 180,E1 -24092.796,E2 -24092.796} C_VEL
LIN {X 0,Y 150.408,Z 506.71,A -85,B 0,C 180,E1 -24094.54,E2 -24094.54} C_VEL
LIN {X 0,Y 150.237,Z 505.817,A -85,B 0,C 180,E1 -24095.746,E2 -24095.746} C_VEL
LIN {X 0,Y 150.356,Z 505.755,A -85,B 0,C 180,E1 -24100.901,E2 -24100.901} C_VEL
LIN {X 0,Y 150.447,Z 505.739,A -85,B 0,C 180,E1 -24106.492,E2 -24106.492} C_VEL
LIN {X 0,Y 150.648,Z 505.695,A -85,B 0,C 180,E1 -24109.245,E2 -24109.245} C_VEL
LIN {X 0,Y 150.742,Z 505.684,A -85,B 0,C 180,E1 -24111.96,E2 -24111.96} C_VEL
LIN {X 0,Y 151.215,Z 505.636,A -85,B 0,C 180,E1 -24120,E2 -24120} C_VEL
LIN {X 0,Y 150.716,Z 505.708,A -85,B 0,C 180,E1 -24128.042,E2 -24128.042} C_VEL
LIN {X 0,Y 150.574,Z 505.702,A -85,B 0,C 180,E1 -24131.437,E2 -24131.437} C_VEL
LIN {X 0,Y 150.376,Z 505.701,A -85,B 0,C 180,E1 -24138.389,E2 -24138.389} C_VEL
LIN {X 0,Y 150.422,Z 506.261,A -85,B 0,C 180,E1 -24139.766,E2 -24139.766} C_VEL
LIN {X 0,Y 152.441,Z 511.834,A -85,B 0,C 180,E1 -24145.608,E2 -24145.608} C_VEL
LIN {X 0,Y 157.133,Z 519.275,A -85,B 0,C 180,E1 -24149.656,E2 -24149.656} C_VEL
LIN {X 0,Y 162.493,Z 528.278,A -85,B 0,C 180,E1 -24153.409,E2 -24153.409} C_VEL
LIN {X 0,Y 166.13,Z 534.724,A -85,B 0,C 180,E1 -24155.662,E2 -24155.662} C_VEL
LIN {X 0,Y 171.652,Z 545.445,A -85,B 0,C 180,E1 -24158.766,E2 -24158.766} C_VEL
LIN {X 0,Y 176.177,Z 555.632,A -85,B 0,C 180,E1 -24161.116,E2 -24161.116} C_VEL
LIN {X 0,Y 180.51,Z 566.639,A -85,B 0,C 180,E1 -24163.236,E2 -24163.236} C_VEL
LIN {X 0,Y 182.022,Z 590.313,A -85,B 0,C 180,E1 -24165.009,E2 -24165.009} C_VEL
LIN {X 0,Y 183.075,Z 616.151,A -85,B 0,C 180,E1 -24166.685,E2 -24166.685} C_VEL
LIN {X 0,Y 181.747,Z 633.235,A -85,B 0,C 180,E1 -24167.364,E2 -24167.364} C_VEL
LIN {X 0,Y 180.022,Z 645.296,A -85,B 0,C 180,E1 -24168.166,E2 -24168.166} C_VEL
LIN {X 0,Y 177.397,Z 657.809,A -85,B 0,C 180,E1 -24169.368,E2 -24169.368} C_VEL
LIN {X 0,Y 174.171,Z 669.546,A -85,B 0,C 180,E1 -24170.915,E2 -24170.915} C_VEL
LIN {X 0,Y 170.283,Z 680.886,A -85,B 0,C 180,E1 -24172.872,E2 -24172.872} C_VEL
LIN {X 0,Y 166.181,Z 691.127,A -85,B 0,C 180,E1 -24175.186,E2 -24175.186} C_VEL
LIN {X 0,Y 162.197,Z 700.404,A -85,B 0,C 180,E1 -24177.942,E2 -24177.942} C_VEL
LIN {X 0,Y 158.016,Z 709.488,A -85,B 0,C 180,E1 -24181.438,E2 -24181.438} C_VEL
LIN {X 0,Y 154.635,Z 716.859,A -85,B 0,C 180,E1 -24185.141,E2 -24185.141} C_VEL
LIN {X 0,Y 152.201,Z 721.846,A -85,B 0,C 180,E1 -24188.322,E2 -24188.322} C_VEL
LIN {X 0,Y 150.354,Z 726.791,A -85,B 0,C 180,E1 -24192.313,E2 -24192.313} C_VEL
LIN {X 0,Y 149.254,Z 730.626,A -85,B 0,C 180,E1 -24196.383,E2 -24196.383} C_VEL
LIN {X 0,Y 148.983,Z 732.647,A -85,B 0,C 180,E1 -24199.124,E2 -24199.124} C_VEL
LIN {X 0,Y 149.027,Z 734.277,A -85,B 0,C 180,E1 -24202.033,E2 -24202.033} C_VEL
LIN {X 0,Y 149.647,Z 735.902,A -85,B 0,C 180,E1 -24206.654,E2 -24206.654} C_VEL
LIN {X 0,Y 149.173,Z 736.12,A -85,B 0,C 180,E1 -24208.135,E2 -24208.135} C_VEL
LIN {X 0,Y 147.672,Z 736.007,A -85,B 0,C 180,E1 -24209.559,E2 -24209.559} C_VEL
LIN {X 0,Y 143.294,Z 735.143,A -85,B 0,C 180,E1 -24212.905,E2 -24212.905} C_VEL
LIN {X 0,Y 142.388,Z 734.628,A -85,B 0,C 180,E1 -24214.498,E2 -24214.498} C_VEL
LIN {X 0,Y 141.964,Z 733.165,A -85,B 0,C 180,E1 -24218.541,E2 -24218.541} C_VEL
LIN {X 0,Y 142.068,Z 730.614,A -85,B 0,C 180,E1 -24222.862,E2 -24222.862} C_VEL
LIN {X 0,Y 143.025,Z 727.09,A -85,B 0,C 180,E1 -24227.147,E2 -24227.147} C_VEL
LIN {X 0,Y 144.844,Z 722.512,A -85,B 0,C 180,E1 -24231.34,E2 -24231.34} C_VEL
LIN {X 0,Y 148.155,Z 715.713,A -85,B 0,C 180,E1 -24236.026,E2 -24236.026} C_VEL
LIN {X 0,Y 151.758,Z 708.306,A -85,B 0,C 180,E1 -24239.856,E2 -24239.856} C_VEL
LIN {X 0,Y 156.205,Z 699.193,A -85,B 0,C 180,E1 -24243.445,E2 -24243.445} C_VEL
LIN {X 0,Y 160.414,Z 689.87,A -85,B 0,C 180,E1 -24246.259,E2 -24246.259} C_VEL
LIN {X 0,Y 164.707,Z 679.556,A -85,B 0,C 180,E1 -24248.611,E2 -24248.611} C_VEL
LIN {X 0,Y 168.656,Z 668.122,A -85,B 0,C 180,E1 -24250.624,E2 -24250.624} C_VEL
LIN {X 0,Y 172.025,Z 656.269,A -85,B 0,C 180,E1 -24252.185,E2 -24252.185} C_VEL
LIN {X 0,Y 174.688,Z 643.868,A -85,B 0,C 180,E1 -24253.368,E2 -24253.368} C_VEL
LIN {X 0,Y 176.636,Z 630.557,A -85,B 0,C 180,E1 -24254.22,E2 -24254.22} C_VEL
LIN {X 0,Y 177.665,Z 616.573,A -85,B 0,C 180,E1 -24254.796,E2 -24254.796} C_VEL
LIN {X 0,Y 176.491,Z 585.16,A -85,B 0,C 180,E1 -24256.934,E2 -24256.934} C_VEL
LIN {X 0,Y 175.405,Z 569.016,A -85,B 0,C 180,E1 -24258.246,E2 -24258.246} C_VEL
LIN {X 0,Y 171.092,Z 557.761,A -85,B 0,C 180,E1 -24260.54,E2 -24260.54} C_VEL
LIN {X 0,Y 166.981,Z 548.499,A -85,B 0,C 180,E1 -24262.849,E2 -24262.849} C_VEL
LIN {X 0,Y 163.855,Z 542.275,A -85,B 0,C 180,E1 -24264.711,E2 -24264.711} C_VEL
LIN {X 0,Y 161.323,Z 537.317,A -85,B 0,C 180,E1 -24266.332,E2 -24266.332} C_VEL
LIN {X 0,Y 157.823,Z 531.075,A -85,B 0,C 180,E1 -24268.731,E2 -24268.731} C_VEL
LIN {X 0,Y 154.18,Z 524.77,A -85,B 0,C 180,E1 -24271.521,E2 -24271.521} C_VEL
LIN {X 0,Y 149.469,Z 517.263,A -85,B 0,C 180,E1 -24275.706,E2 -24275.706} C_VEL
LIN {X 0,Y 144.391,Z 509.634,A -85,B 0,C 180,E1 -24281.556,E2 -24281.556} C_VEL
LIN {X 0,Y 143.4,Z 507.144,A -85,B 0,C 180,E1 -24284.362,E2 -24284.362} C_VEL
LIN {X 0,Y 143.355,Z 506.682,A -85,B 0,C 180,E1 -24285.811,E2 -24285.811} C_VEL
LIN {X 0,Y 143.534,Z 506.578,A -85,B 0,C 180,E1 -24288.705,E2 -24288.705} C_VEL
LIN {X 0,Y 143.634,Z 506.585,A -85,B 0,C 180,E1 -24291.559,E2 -24291.559} C_VEL
LIN {X 0,Y 144.174,Z 506.515,A -85,B 0,C 180,E1 -24300,E2 -24300} C_VEL
LIN {X 0,Y 143.623,Z 506.568,A -85,B 0,C 180,E1 -24308.442,E2 -24308.442} C_VEL
LIN {X 0,Y 143.501,Z 506.593,A -85,B 0,C 180,E1 -24311.627,E2 -24311.627} C_VEL
LIN {X 0,Y 143.306,Z 506.882,A -85,B 0,C 180,E1 -24318.034,E2 -24318.034} C_VEL
LIN {X 0,Y 143.583,Z 507.866,A -85,B 0,C 180,E1 -24319.293,E2 -24319.293} C_VEL
LIN {X 0,Y 145.177,Z 510.677,A -85,B 0,C 180,E1 -24321.568,E2 -24321.568} C_VEL
LIN {X 0,Y 148.163,Z 512.821,A -85,B 0,C 180,E1 -24324.709,E2 -24324.709} C_VEL
LIN {X 0,Y 150.046,Z 516.084,A -85,B 0,C 180,E1 -24326.653,E2 -24326.653} C_VEL
LIN {X 0,Y 152.621,Z 518.337,A -85,B 0,C 180,E1 -24328.822,E2 -24328.822} C_VEL
LIN {X 0,Y 154.923,Z 521.791,A -85,B 0,C 180,E1 -24330.713,E2 -24330.713} C_VEL
LIN {X 0,Y 156.59,Z 523.587,A -85,B 0,C 180,E1 -24331.923,E2 -24331.923} C_VEL
LIN {X 0,Y 159.34,Z 527.274,A -85,B 0,C 180,E1 -24333.839,E2 -24333.839} C_VEL
LIN {X 0,Y 163.78,Z 533.624,A -85,B 0,C 180,E1 -24336.644,E2 -24336.644} C_VEL
LIN {X 0,Y 168.825,Z 541.187,A -85,B 0,C 180,E1 -24339.477,E2 -24339.477} C_VEL
LIN {X 0,Y 174.258,Z 550.245,A -85,B 0,C 180,E1 -24342.231,E2 -24342.231} C_VEL
LIN {X 0,Y 179.807,Z 560.794,A -85,B 0,C 180,E1 -24344.811,E2 -24344.811} C_VEL
LIN {X 0,Y 181.116,Z 563.638,A -85,B 0,C 180,E1 -24345.399,E2 -24345.399} C_VEL
LIN {X 0,Y 179.736,Z 593.634,A -85,B 0,C 180,E1 -24346.717,E2 -24346.717} C_VEL
LIN {X 0,Y 178.346,Z 606.833,A -85,B 0,C 180,E1 -24347.698,E2 -24347.698} C_VEL
LIN {X 0,Y 176.378,Z 618.342,A -85,B 0,C 180,E1 -24348.896,E2 -24348.896} C_VEL
LIN {X 0,Y 173.722,Z 629.871,A -85,B 0,C 180,E1 -24350.507,E2 -24350.507} C_VEL
LIN {X 0,Y 170.294,Z 641.018,A -85,B 0,C 180,E1 -24352.503,E2 -24352.503} C_VEL
LIN {X 0,Y 166.61,Z 651.327,A -85,B 0,C 180,E1 -24354.92,E2 -24354.92} C_VEL
LIN {X 0,Y 163.198,Z 659.731,A -85,B 0,C 180,E1 -24357.433,E2 -24357.433} C_VEL
LIN {X 0,Y 159.751,Z 667.452,A -85,B 0,C 180,E1 -24360.336,E2 -24360.336} C_VEL
LIN {X 0,Y 155.858,Z 675.112,A -85,B 0,C 180,E1 -24363.991,E2 -24363.991} C_VEL
LIN {X 0,Y 152.16,Z 681.909,A -85,B 0,C 180,E1 -24368.315,E2 -24368.315} C_VEL
LIN {X 0,Y 149.418,Z 686.513,A -85,B 0,C 180,E1 -24372.198,E2 -24372.198} C_VEL
LIN {X 0,Y 147.115,Z 690.047,A -85,B 0,C 180,E1 -24376.181,E2 -24376.181} C_VEL
LIN {X 0,Y 145.937,Z 691.868,A -85,B 0,C 180,E1 -24378.894,E2 -24378.894} C_VEL
LIN {X 0,Y 144.78,Z 694.147,A -85,B 0,C 180,E1 -24384.429,E2 -24384.429} C_VEL
LIN {X 0,Y 144.223,Z 694.972,A -85,B 0,C 180,E1 -24390,E2 -24390} C_VEL
LIN {X 0,Y 144.776,Z 694.196,A -85,B 0,C 180,E1 -24395.571,E2 -24395.571} C_VEL
LIN {X 0,Y 145.919,Z 691.969,A -85,B 0,C 180,E1 -24401.107,E2 -24401.107} C_VEL
LIN {X 0,Y 147.864,Z 689.135,A -85,B 0,C 180,E1 -24405.154,E2 -24405.154} C_VEL
LIN {X 0,Y 150.329,Z 685.3,A -85,B 0,C 180,E1 -24409.102,E2 -24409.102} C_VEL
LIN {X 0,Y 153.176,Z 680.211,A -85,B 0,C 180,E1 -24413.095,E2 -24413.095} C_VEL
LIN {X 0,Y 156.492,Z 674.169,A -85,B 0,C 180,E1 -24416.685,E2 -24416.685} C_VEL
LIN {X 0,Y 160.406,Z 666.378,A -85,B 0,C 180,E1 -24420.255,E2 -24420.255} C_VEL
LIN {X 0,Y 164.634,Z 656.694,A -85,B 0,C 180,E1 -24423.706,E2 -24423.706} C_VEL
LIN {X 0,Y 168.164,Z 647.631,A -85,B 0,C 180,E1 -24426.179,E2 -24426.179} C_VEL
LIN {X 0,Y 171.793,Z 637.094,A -85,B 0,C 180,E1 -24428.393,E2 -24428.393} C_VEL
LIN {X 0,Y 175.01,Z 625.389,A -85,B 0,C 180,E1 -24430.317,E2 -24430.317} C_VEL
LIN {X 0,Y 177.554,Z 613.875,A -85,B 0,C 180,E1 -24431.717,E2 -24431.717} C_VEL
LIN {X 0,Y 179.269,Z 600.844,A -85,B 0,C 180,E1 -24432.939,E2 -24432.939} C_VEL
LIN {X 0,Y 180.222,Z 588.733,A -85,B 0,C 180,E1 -24433.681,E2 -24433.681} C_VEL
LIN {X 0,Y 181.273,Z 563.817,A -85,B 0,C 180,E1 -24434.742,E2 -24434.742} C_VEL
LIN {X 0,Y 176.637,Z 554.504,A -85,B 0,C 180,E1 -24436.854,E2 -24436.854} C_VEL
LIN {X 0,Y 171.095,Z 544.813,A -85,B 0,C 180,E1 -24439.568,E2 -24439.568} C_VEL
LIN {X 0,Y 165.21,Z 535.51,A -85,B 0,C 180,E1 -24442.781,E2 -24442.781} C_VEL
LIN {X 0,Y 161.832,Z 530.808,A -85,B 0,C 180,E1 -24444.806,E2 -24444.806} C_VEL
LIN {X 0,Y 159.045,Z 526.907,A -85,B 0,C 180,E1 -24446.632,E2 -24446.632} C_VEL
LIN {X 0,Y 156.559,Z 523.416,A -85,B 0,C 180,E1 -24448.402,E2 -24448.402} C_VEL
LIN {X 0,Y 153.176,Z 519.291,A -85,B 0,C 180,E1 -24451.012,E2 -24451.012} C_VEL
LIN {X 0,Y 152.304,Z 517.929,A -85,B 0,C 180,E1 -24451.772,E2 -24451.772} C_VEL
LIN {X 0,Y 149.772,Z 515.708,A -85,B 0,C 180,E1 -24453.961,E2 -24453.961} C_VEL
LIN {X 0,Y 148.022,Z 512.571,A -85,B 0,C 180,E1 -24455.826,E2 -24455.826} C_VEL
LIN {X 0,Y 145.159,Z 510.622,A -85,B 0,C 180,E1 -24458.894,E2 -24458.894} C_VEL
LIN {X 0,Y 143.637,Z 508.02,A -85,B 0,C 180,E1 -24461.086,E2 -24461.086} C_VEL
LIN {X 0,Y 143.315,Z 506.898,A -85,B 0,C 180,E1 -24462.52,E2 -24462.52} C_VEL
LIN {X 0,Y 143.592,Z 506.578,A -85,B 0,C 180,E1 -24468.71,E2 -24468.71} C_VEL
LIN {X 0,Y 143.661,Z 506.562,A -85,B 0,C 180,E1 -24471.56,E2 -24471.56} C_VEL
LIN {X 0,Y 144.174,Z 506.511,A -85,B 0,C 180,E1 -24480,E2 -24480} C_VEL
LIN {X 0,Y 143.634,Z 506.582,A -85,B 0,C 180,E1 -24488.441,E2 -24488.441} C_VEL
LIN {X 0,Y 143.502,Z 506.583,A -85,B 0,C 180,E1 -24491.629,E2 -24491.629} C_VEL
LIN {X 0,Y 143.342,Z 506.858,A -85,B 0,C 180,E1 -24494.916,E2 -24494.916} C_VEL
LIN {X 0,Y 144.183,Z 509.172,A -85,B 0,C 180,E1 -24497.737,E2 -24497.737} C_VEL
LIN {X 0,Y 150.359,Z 518.449,A -85,B 0,C 180,E1 -24504.877,E2 -24504.877} C_VEL
LIN {X 0,Y 154.675,Z 525.323,A -85,B 0,C 180,E1 -24508.643,E2 -24508.643} C_VEL
LIN {X 0,Y 159.428,Z 533.746,A -85,B 0,C 180,E1 -24512.208,E2 -24512.208} C_VEL
LIN {X 0,Y 162.871,Z 540.148,A -85,B 0,C 180,E1 -24514.496,E2 -24514.496} C_VEL
LIN {X 0,Y 166.514,Z 547.465,A -85,B 0,C 180,E1 -24516.728,E2 -24516.728} C_VEL
LIN {X 0,Y 170.504,Z 556.118,A -85,B 0,C 180,E1 -24518.99,E2 -24518.99} C_VEL
LIN {X 0,Y 174.954,Z 567.406,A -85,B 0,C 180,E1 -24521.377,E2 -24521.377} C_VEL
LIN {X 0,Y 175.769,Z 570.313,A -85,B 0,C 180,E1 -24521.84,E2 -24521.84} C_VEL
LIN {X 0,Y 177.125,Z 596.004,A -85,B 0,C 180,E1 -24523.78,E2 -24523.78} C_VEL
LIN {X 0,Y 177.83,Z 617.453,A -85,B 0,C 180,E1 -24525.197,E2 -24525.197} C_VEL
LIN {X 0,Y 176.55,Z 632.575,A -85,B 0,C 180,E1 -24525.82,E2 -24525.82} C_VEL
LIN {X 0,Y 174.724,Z 644.506,A -85,B 0,C 180,E1 -24526.617,E2 -24526.617} C_VEL
LIN {X 0,Y 172.068,Z 656.817,A -85,B 0,C 180,E1 -24527.828,E2 -24527.828} C_VEL
LIN {X 0,Y 168.684,Z 668.546,A -85,B 0,C 180,E1 -24529.385,E2 -24529.385} C_VEL
LIN {X 0,Y 164.682,Z 679.893,A -85,B 0,C 180,E1 -24531.382,E2 -24531.382} C_VEL
LIN {X 0,Y 160.401,Z 690.131,A -85,B 0,C 180,E1 -24533.737,E2 -24533.737} C_VEL
LIN {X 0,Y 156.175,Z 699.4,A -85,B 0,C 180,E1 -24536.548,E2 -24536.548} C_VEL
LIN {X 0,Y 151.762,Z 708.483,A -85,B 0,C 180,E1 -24540.145,E2 -24540.145} C_VEL
LIN {X 0,Y 148.158,Z 715.852,A -85,B 0,C 180,E1 -24543.974,E2 -24543.974} C_VEL
LIN {X 0,Y 144.776,Z 722.605,A -85,B 0,C 180,E1 -24548.65,E2 -24548.65} C_VEL
LIN {X 0,Y 143.014,Z 727.167,A -85,B 0,C 180,E1 -24552.852,E2 -24552.852} C_VEL
LIN {X 0,Y 142.066,Z 730.667,A -85,B 0,C 180,E1 -24557.138,E2 -24557.138} C_VEL
LIN {X 0,Y 141.969,Z 733.402,A -85,B 0,C 180,E1 -24561.921,E2 -24561.921} C_VEL
LIN {X 0,Y 142.704,Z 735.083,A -85,B 0,C 180,E1 -24567.177,E2 -24567.177} C_VEL
LIN {X 0,Y 143.376,Z 735.41,A -85,B 0,C 180,E1 -24570,E2 -24570} C_VEL
LIN {X 0,Y 142.388,Z 734.628,A -85,B 0,C 180,E1 -24574.498,E2 -24574.498} C_VEL
LIN {X 0,Y 141.42,Z 733.843,A -85,B 0,C 180,E1 -24576.829,E2 -24576.829} C_VEL
LIN {X 0,Y 138.405,Z 731.825,A -85,B 0,C 180,E1 -24580.617,E2 -24580.617} C_VEL
LIN {X 0,Y 136.243,Z 729.688,A -85,B 0,C 180,E1 -24583.701,E2 -24583.701} C_VEL
LIN {X 0,Y 135.675,Z 727.802,A -85,B 0,C 180,E1 -24586.065,E2 -24586.065} C_VEL
LIN {X 0,Y 135.808,Z 727.127,A -85,B 0,C 180,E1 -24586.849,E2 -24586.849} C_VEL
LIN {X 0,Y 137.444,Z 723.179,A -85,B 0,C 180,E1 -24590.973,E2 -24590.973} C_VEL
LIN {X 0,Y 140.694,Z 716.769,A -85,B 0,C 180,E1 -24595.954,E2 -24595.954} C_VEL
LIN {X 0,Y 144.244,Z 709.932,A -85,B 0,C 180,E1 -24599.96,E2 -24599.96} C_VEL
LIN {X 0,Y 148.676,Z 701.471,A -85,B 0,C 180,E1 -24603.739,E2 -24603.739} C_VEL
LIN {X 0,Y 152.885,Z 692.823,A -85,B 0,C 180,E1 -24606.697,E2 -24606.697} C_VEL
LIN {X 0,Y 157.675,Z 682.211,A -85,B 0,C 180,E1 -24609.431,E2 -24609.431} C_VEL
LIN {X 0,Y 161.791,Z 671.733,A -85,B 0,C 180,E1 -24611.485,E2 -24611.485} C_VEL
LIN {X 0,Y 165.447,Z 660.226,A -85,B 0,C 180,E1 -24613.232,E2 -24613.232} C_VEL
LIN {X 0,Y 168.483,Z 648.385,A -85,B 0,C 180,E1 -24614.53,E2 -24614.53} C_VEL
LIN {X 0,Y 170.939,Z 634.743,A -85,B 0,C 180,E1 -24615.588,E2 -24615.588} C_VEL
LIN {X 0,Y 172.385,Z 621.465,A -85,B 0,C 180,E1 -24616.218,E2 -24616.218} C_VEL
LIN {X 0,Y 172.527,Z 614.537,A -85,B 0,C 180,E1 -24616.573,E2 -24616.573} C_VEL
LIN {X 0,Y 171.446,Z 582.906,A -85,B 0,C 180,E1 -24618.841,E2 -24618.841} C_VEL
LIN {X 0,Y 170.748,Z 571.926,A -85,B 0,C 180,E1 -24619.782,E2 -24619.782} C_VEL
LIN {X 0,Y 166.515,Z 560.62,A -85,B 0,C 180,E1 -24622.229,E2 -24622.229} C_VEL
LIN {X 0,Y 162.283,Z 551.028,A -85,B 0,C 180,E1 -24624.826,E2 -24624.826} C_VEL
LIN {X 0,Y 158.185,Z 542.638,A -85,B 0,C 180,E1 -24627.579,E2 -24627.579} C_VEL
LIN {X 0,Y 154.759,Z 536.337,A -85,B 0,C 180,E1 -24630.105,E2 -24630.105} C_VEL
LIN {X 0,Y 151.475,Z 530.413,A -85,B 0,C 180,E1 -24632.824,E2 -24632.824} C_VEL
LIN {X 0,Y 147.464,Z 523.613,A -85,B 0,C 180,E1 -24636.661,E2 -24636.661} C_VEL
LIN {X 0,Y 142.574,Z 515.966,A -85,B 0,C 180,E1 -24642.612,E2 -24642.612} C_VEL
LIN {X 0,Y 140.712,Z 513.299,A -85,B 0,C 180,E1 -24645.539,E2 -24645.539} C_VEL
LIN {X 0,Y 137.164,Z 509.617,A -85,B 0,C 180,E1 -24653.749,E2 -24653.749} C_VEL
LIN {X 0,Y 136.859,Z 508.039,A -85,B 0,C 180,E1 -24657.057,E2 -24657.057} C_VEL
LIN {X 0,Y 137.152,Z 507.555,A -85,B 0,C 180,E1 -24660,E2 -24660} C_VEL
LIN {X 0,Y 136.752,Z 508.39,A -85,B 0,C 180,E1 -24665.53,E2 -24665.53} C_VEL
LIN {X 0,Y 137.676,Z 510.582,A -85,B 0,C 180,E1 -24670.106,E2 -24670.106} C_VEL
LIN {X 0,Y 140.185,Z 513.024,A -85,B 0,C 180,E1 -24675.633,E2 -24675.633} C_VEL
LIN {X 0,Y 141.749,Z 513.999,A -85,B 0,C 180,E1 -24678.052,E2 -24678.052} C_VEL
LIN {X 0,Y 143.434,Z 517.105,A -85,B 0,C 180,E1 -24680.587,E2 -24680.587} C_VEL
LIN {X 0,Y 146.305,Z 519.507,A -85,B 0,C 180,E1 -24683.836,E2 -24683.836} C_VEL
LIN {X 0,Y 148.369,Z 522.831,A -85,B 0,C 180,E1 -24686.036,E2 -24686.036} C_VEL
LIN {X 0,Y 150.553,Z 524.953,A -85,B 0,C 180,E1 -24687.981,E2 -24687.981} C_VEL
LIN {X 0,Y 153.073,Z 528.49,A -85,B 0,C 180,E1 -24690.115,E2 -24690.115} C_VEL
LIN {X 0,Y 154.34,Z 530.112,A -85,B 0,C 180,E1 -24691.097,E2 -24691.097} C_VEL
LIN {X 0,Y 157.853,Z 535.034,A -85,B 0,C 180,E1 -24693.639,E2 -24693.639} C_VEL
LIN {X 0,Y 161.172,Z 539.826,A -85,B 0,C 180,E1 -24695.806,E2 -24695.806} C_VEL
LIN {X 0,Y 166.684,Z 548.526,A -85,B 0,C 180,E1 -24699.047,E2 -24699.047} C_VEL
LIN {X 0,Y 172.084,Z 558.171,A -85,B 0,C 180,E1 -24701.896,E2 -24701.896} C_VEL
LIN {X 0,Y 176.126,Z 566.364,A -85,B 0,C 180,E1 -24703.875,E2 -24703.875} C_VEL
LIN {X 0,Y 174.694,Z 594.513,A -85,B 0,C 180,E1 -24705.128,E2 -24705.128} C_VEL
LIN {X 0,Y 173.183,Z 608.011,A -85,B 0,C 180,E1 -24706.147,E2 -24706.147} C_VEL
LIN {X 0,Y 171.144,Z 619.337,A -85,B 0,C 180,E1 -24707.349,E2 -24707.349} C_VEL
LIN {X 0,Y 168.465,Z 630.475,A -85,B 0,C 180,E1 -24708.92,E2 -24708.92} C_VEL
LIN {X 0,Y 164.773,Z 642.01,A -85,B 0,C 180,E1 -24711.015,E2 -24711.015} C_VEL
LIN {X 0,Y 160.908,Z 652.319,A -85,B 0,C 180,E1 -24713.481,E2 -24713.481} C_VEL
LIN {X 0,Y 157.32,Z 660.722,A -85,B 0,C 180,E1 -24716.055,E2 -24716.055} C_VEL
LIN {X 0,Y 153.683,Z 668.442,A -85,B 0,C 180,E1 -24719.039,E2 -24719.039} C_VEL
LIN {X 0,Y 149.573,Z 676.102,A -85,B 0,C 180,E1 -24722.81,E2 -24722.81} C_VEL
LIN {X 0,Y 145.653,Z 682.898,A -85,B 0,C 180,E1 -24727.294,E2 -24727.294} C_VEL
LIN {X 0,Y 142.742,Z 687.502,A -85,B 0,C 180,E1 -24731.336,E2 -24731.336} C_VEL
LIN {X 0,Y 140.299,Z 691.037,A -85,B 0,C 180,E1 -24735.495,E2 -24735.495} C_VEL
LIN {X 0,Y 139.045,Z 692.857,A -85,B 0,C 180,E1 -24738.336,E2 -24738.336} C_VEL
LIN {X 0,Y 137.787,Z 695.135,A -85,B 0,C 180,E1 -24744.145,E2 -24744.145} C_VEL
LIN {X 0,Y 137.195,Z 695.96,A -85,B 0,C 180,E1 -24750,E2 -24750} C_VEL
LIN {X 0,Y 137.783,Z 695.184,A -85,B 0,C 180,E1 -24755.855,E2 -24755.855} C_VEL
LIN {X 0,Y 139.026,Z 692.957,A -85,B 0,C 180,E1 -24761.666,E2 -24761.666} C_VEL
LIN {X 0,Y 141.092,Z 690.122,A -85,B 0,C 180,E1 -24765.9,E2 -24765.9} C_VEL
LIN {X 0,Y 143.707,Z 686.287,A -85,B 0,C 180,E1 -24770.019,E2 -24770.019} C_VEL
LIN {X 0,Y 146.738,Z 681.198,A -85,B 0,C 180,E1 -24774.172,E2 -24774.172} C_VEL
LIN {X 0,Y 150.246,Z 675.155,A -85,B 0,C 180,E1 -24777.889,E2 -24777.889} C_VEL
LIN {X 0,Y 154.376,Z 667.363,A -85,B 0,C 180,E1 -24781.569,E2 -24781.569} C_VEL
LIN {X 0,Y 158.834,Z 657.679,A -85,B 0,C 180,E1 -24785.114,E2 -24785.114} C_VEL
LIN {X 0,Y 162.525,Z 648.619,A -85,B 0,C 180,E1 -24787.646,E2 -24787.646} C_VEL
LIN {X 0,Y 166.689,Z 637.055,A -85,B 0,C 180,E1 -24790.083,E2 -24790.083} C_VEL
LIN {X 0,Y 169.967,Z 625.407,A -85,B 0,C 180,E1 -24791.994,E2 -24791.994} C_VEL
LIN {X 0,Y 172.599,Z 613.587,A -85,B 0,C 180,E1 -24793.401,E2 -24793.401} C_VEL
LIN {X 0,Y 174.29,Z 600.935,A -85,B 0,C 180,E1 -24794.581,E2 -24794.581} C_VEL
LIN {X 0,Y 175.282,Z 588.275,A -85,B 0,C 180,E1 -24795.341,E2 -24795.341} C_VEL
LIN {X 0,Y 176.272,Z 566.507,A -85,B 0,C 180,E1 -24796.275,E2 -24796.275} C_VEL
LIN {X 0,Y 171.935,Z 557.801,A -85,B 0,C 180,E1 -24798.406,E2 -24798.406} C_VEL
LIN {X 0,Y 166.387,Z 547.903,A -85,B 0,C 180,E1 -24801.366,E2 -24801.366} C_VEL
LIN {X 0,Y 159.844,Z 537.601,A -85,B 0,C 180,E1 -24805.326,E2 -24805.326} C_VEL
LIN {X 0,Y 156.215,Z 532.677,A -85,B 0,C 180,E1 -24807.802,E2 -24807.802} C_VEL
LIN {X 0,Y 153.435,Z 528.721,A -85,B 0,C 180,E1 -24809.929,E2 -24809.929} C_VEL
LIN {X 0,Y 150.722,Z 525.153,A -85,B 0,C 180,E1 -24812.206,E2 -24812.206} C_VEL
LIN {X 0,Y 149.924,Z 524.218,A -85,B 0,C 180,E1 -24812.915,E2 -24812.915} C_VEL
LIN {X 0,Y 147.415,Z 521.521,A -85,B 0,C 180,E1 -24815.298,E2 -24815.298} C_VEL
LIN {X 0,Y 145.934,Z 519.099,A -85,B 0,C 180,E1 -24816.965,E2 -24816.965} C_VEL
LIN {X 0,Y 143.463,Z 517.092,A -85,B 0,C 180,E1 -24819.84,E2 -24819.84} C_VEL
LIN {X 0,Y 141.78,Z 514.063,A -85,B 0,C 180,E1 -24822.418,E2 -24822.418} C_VEL
LIN {X 0,Y 140.117,Z 512.951,A -85,B 0,C 180,E1 -24825.104,E2 -24825.104} C_VEL
LIN {X 0,Y 136.859,Z 508.331,A -85,B 0,C 180,E1 -24836.319,E2 -24836.319} C_VEL
LIN {X 0,Y 137.174,Z 507.745,A -85,B 0,C 180,E1 -24840,E2 -24840} C_VEL
LIN {X 0,Y 136.997,Z 508.828,A -85,B 0,C 180,E1 -24843.677,E2 -24843.677} C_VEL
LIN {X 0,Y 140.568,Z 513.216,A -85,B 0,C 180,E1 -24853.738,E2 -24853.738} C_VEL
LIN {X 0,Y 141.503,Z 514.23,A -85,B 0,C 180,E1 -24855.299,E2 -24855.299} C_VEL
LIN {X 0,Y 143.659,Z 517.701,A -85,B 0,C 180,E1 -24858.541,E2 -24858.541} C_VEL
LIN {X 0,Y 148.317,Z 524.921,A -85,B 0,C 180,E1 -24863.937,E2 -24863.937} C_VEL
LIN {X 0,Y 152.687,Z 532.343,A -85,B 0,C 180,E1 -24867.977,E2 -24867.977} C_VEL
LIN {X 0,Y 156.49,Z 539.33,A -85,B 0,C 180,E1 -24871.002,E2 -24871.002} C_VEL
LIN {X 0,Y 159.696,Z 545.568,A -85,B 0,C 180,E1 -24873.291,E2 -24873.291} C_VEL
LIN {X 0,Y 164.03,Z 554.51,A -85,B 0,C 180,E1 -24876.095,E2 -24876.095} C_VEL
LIN {X 0,Y 167.988,Z 564.123,A -85,B 0,C 180,E1 -24878.485,E2 -24878.485} C_VEL
LIN {X 0,Y 170.977,Z 572.327,A -85,B 0,C 180,E1 -24880.203,E2 -24880.203} C_VEL
LIN {X 0,Y 172.076,Z 594.344,A -85,B 0,C 180,E1 -24881.958,E2 -24881.958} C_VEL
LIN {X 0,Y 172.754,Z 617.863,A -85,B 0,C 180,E1 -24883.581,E2 -24883.581} C_VEL
LIN {X 0,Y 171.391,Z 632.623,A -85,B 0,C 180,E1 -24884.215,E2 -24884.215} C_VEL
LIN {X 0,Y 169.287,Z 645.187,A -85,B 0,C 180,E1 -24885.111,E2 -24885.111} C_VEL
LIN {X 0,Y 166.588,Z 656.821,A -85,B 0,C 180,E1 -24886.306,E2 -24886.306} C_VEL
LIN {X 0,Y 163.334,Z 667.548,A -85,B 0,C 180,E1 -24887.755,E2 -24887.755} C_VEL
LIN {X 0,Y 159.202,Z 678.9,A -85,B 0,C 180,E1 -24889.789,E2 -24889.789} C_VEL
LIN {X 0,Y 154.738,Z 689.137,A -85,B 0,C 180,E1 -24892.183,E2 -24892.183} C_VEL
LIN {X 0,Y 150.262,Z 698.398,A -85,B 0,C 180,E1 -24895.045,E2 -24895.045} C_VEL
LIN {X 0,Y 145.603,Z 707.479,A -85,B 0,C 180,E1 -24898.744,E2 -24898.744} C_VEL
LIN {X 0,Y 141.762,Z 714.848,A -85,B 0,C 180,E1 -24902.705,E2 -24902.705} C_VEL
LIN {X 0,Y 138.124,Z 721.599,A -85,B 0,C 180,E1 -24907.567,E2 -24907.567} C_VEL
LIN {X 0,Y 136.174,Z 726.159,A -85,B 0,C 180,E1 -24911.962,E2 -24911.962} C_VEL
LIN {X 0,Y 135.091,Z 729.66,A -85,B 0,C 180,E1 -24916.461,E2 -24916.461} C_VEL
LIN {X 0,Y 134.91,Z 732.529,A -85,B 0,C 180,E1 -24921.804,E2 -24921.804} C_VEL
LIN {X 0,Y 135.618,Z 734.085,A -85,B 0,C 180,E1 -24927.03,E2 -24927.03} C_VEL
LIN {X 0,Y 136.291,Z 734.413,A -85,B 0,C 180,E1 -24930,E2 -24930} C_VEL
LIN {X 0,Y 135.368,Z 733.749,A -85,B 0,C 180,E1 -24934.249,E2 -24934.249} C_VEL
LIN {X 0,Y 134.899,Z 732.159,A -85,B 0,C 180,E1 -24938.992,E2 -24938.992} C_VEL
LIN {X 0,Y 135.093,Z 729.606,A -85,B 0,C 180,E1 -24943.539,E2 -24943.539} C_VEL
LIN {X 0,Y 135.808,Z 727.127,A -85,B 0,C 180,E1 -24946.849,E2 -24946.849} C_VEL
LIN {X 0,Y 135.632,Z 725.724,A -85,B 0,C 180,E1 -24948.425,E2 -24948.425} C_VEL
LIN {X 0,Y 132.25,Z 720.535,A -85,B 0,C 180,E1 -24953.574,E2 -24953.574} C_VEL
LIN {X 0,Y 132.583,Z 718.716,A -85,B 0,C 180,E1 -24955.098,E2 -24955.098} C_VEL
LIN {X 0,Y 136.716,Z 711.394,A -85,B 0,C 180,E1 -24960.079,E2 -24960.079} C_VEL
LIN {X 0,Y 141.141,Z 703.494,A -85,B 0,C 180,E1 -24964.067,E2 -24964.067} C_VEL
LIN {X 0,Y 146.313,Z 693.653,A -85,B 0,C 180,E1 -24967.764,E2 -24967.764} C_VEL
LIN {X 0,Y 151.213,Z 683.554,A -85,B 0,C 180,E1 -24970.592,E2 -24970.592} C_VEL
LIN {X 0,Y 155.986,Z 672.164,A -85,B 0,C 180,E1 -24972.956,E2 -24972.956} C_VEL
LIN {X 0,Y 159.778,Z 661.003,A -85,B 0,C 180,E1 -24974.729,E2 -24974.729} C_VEL
LIN {X 0,Y 163.201,Z 648.642,A -85,B 0,C 180,E1 -24976.161,E2 -24976.161} C_VEL
LIN {X 0,Y 165.812,Z 635.195,A -85,B 0,C 180,E1 -24977.248,E2 -24977.248} C_VEL
LIN {X 0,Y 167.288,Z 623.33,A -85,B 0,C 180,E1 -24977.862,E2 -24977.862} C_VEL
LIN {X 0,Y 167.624,Z 616.167,A -85,B 0,C 180,E1 -24978.208,E2 -24978.208} C_VEL
LIN {X 0,Y 166.657,Z 582.724,A -85,B 0,C 180,E1 -24980.704,E2 -24980.704} C_VEL
LIN {X 0,Y 166.175,Z 574.607,A -85,B 0,C 180,E1 -24981.436,E2 -24981.436} C_VEL
LIN {X 0,Y 161.804,Z 562.812,A -85,B 0,C 180,E1 -24984.196,E2 -24984.196} C_VEL
LIN {X 0,Y 157.545,Z 553.137,A -85,B 0,C 180,E1 -24987.084,E2 -24987.084} C_VEL
LIN {X 0,Y 154.528,Z 546.9,A -85,B 0,C 180,E1 -24989.321,E2 -24989.321} C_VEL
LIN {X 0,Y 151.834,Z 541.648,A -85,B 0,C 180,E1 -24991.498,E2 -24991.498} C_VEL
LIN {X 0,Y 149.005,Z 536.238,A -85,B 0,C 180,E1 -24994.039,E2 -24994.039} C_VEL
LIN {X 0,Y 145.22,Z 529.554,A -85,B 0,C 180,E1 -24997.952,E2 -24997.952} C_VEL
LIN {X 0,Y 140.882,Z 522.338,A -85,B 0,C 180,E1 -25003.704,E2 -25003.704} C_VEL
LIN {X 0,Y 139.436,Z 520.157,A -85,B 0,C 180,E1 -25006.148,E2 -25006.148} C_VEL
LIN {X 0,Y 136.119,Z 516.444,A -85,B 0,C 180,E1 -25014.445,E2 -25014.445} C_VEL
LIN {X 0,Y 135.634,Z 514.888,A -85,B 0,C 180,E1 -25017.773,E2 -25017.773} C_VEL
LIN {X 0,Y 135.489,Z 514.472,A -85,B 0,C 180,E1 -25020,E2 -25020} C_VEL
LIN {X 0,Y 135.768,Z 515.529,A -85,B 0,C 180,E1 -25025.57,E2 -25025.57} C_VEL
LIN {X 0,Y 138.741,Z 519.773,A -85,B 0,C 180,E1 -25034.672,E2 -25034.672} C_VEL
LIN {X 0,Y 140.215,Z 520.673,A -85,B 0,C 180,E1 -25037.126,E2 -25037.126} C_VEL
LIN {X 0,Y 142.085,Z 524.017,A -85,B 0,C 180,E1 -25040.071,E2 -25040.071} C_VEL
LIN {X 0,Y 144.463,Z 526.059,A -85,B 0,C 180,E1 -25042.905,E2 -25042.905} C_VEL
LIN {X 0,Y 146.652,Z 529.489,A -85,B 0,C 180,E1 -25045.345,E2 -25045.345} C_VEL
LIN {X 0,Y 148.423,Z 531.357,A -85,B 0,C 180,E1 -25047.018,E2 -25047.018} C_VEL
LIN {X 0,Y 151.165,Z 535.091,A -85,B 0,C 180,E1 -25049.44,E2 -25049.44} C_VEL
LIN {X 0,Y 155.431,Z 541.292,A -85,B 0,C 180,E1 -25052.759,E2 -25052.759} C_VEL
LIN {X 0,Y 159.397,Z 547.339,A -85,B 0,C 180,E1 -25055.468,E2 -25055.468} C_VEL
LIN {X 0,Y 165.112,Z 556.912,A -85,B 0,C 180,E1 -25058.929,E2 -25058.929} C_VEL
LIN {X 0,Y 170.364,Z 567.205,A -85,B 0,C 180,E1 -25061.797,E2 -25061.797} C_VEL
LIN {X 0,Y 171.165,Z 568.84,A -85,B 0,C 180,E1 -25062.209,E2 -25062.209} C_VEL
LIN {X 0,Y 169.764,Z 595.99,A -85,B 0,C 180,E1 -25063.493,E2 -25063.493} C_VEL
LIN {X 0,Y 168.152,Z 609.205,A -85,B 0,C 180,E1 -25064.505,E2 -25064.505} C_VEL
LIN {X 0,Y 165.817,Z 621.497,A -85,B 0,C 180,E1 -25065.862,E2 -25065.862} C_VEL
LIN {X 0,Y 162.888,Z 632.643,A -85,B 0,C 180,E1 -25067.502,E2 -25067.502} C_VEL
LIN {X 0,Y 159.37,Z 643.003,A -85,B 0,C 180,E1 -25069.425,E2 -25069.425} C_VEL
LIN {X 0,Y 155.316,Z 653.311,A -85,B 0,C 180,E1 -25071.938,E2 -25071.938} C_VEL
LIN {X 0,Y 151.541,Z 661.713,A -85,B 0,C 180,E1 -25074.571,E2 -25074.571} C_VEL
LIN {X 0,Y 147.7,Z 669.433,A -85,B 0,C 180,E1 -25077.636,E2 -25077.636} C_VEL
LIN {X 0,Y 143.358,Z 677.092,A -85,B 0,C 180,E1 -25081.527,E2 -25081.527} C_VEL
LIN {X 0,Y 139.196,Z 683.888,A -85,B 0,C 180,E1 -25086.177,E2 -25086.177} C_VEL
LIN {X 0,Y 136.102,Z 688.491,A -85,B 0,C 180,E1 -25090.389,E2 -25090.389} C_VEL
LIN {X 0,Y 133.505,Z 692.026,A -85,B 0,C 180,E1 -25094.74,E2 -25094.74} C_VEL
LIN {X 0,Y 132.167,Z 693.846,A -85,B 0,C 180,E1 -25097.72,E2 -25097.72} C_VEL
LIN {X 0,Y 130.797,Z 696.124,A -85,B 0,C 180,E1 -25103.831,E2 -25103.831} C_VEL
LIN {X 0,Y 130.167,Z 696.948,A -85,B 0,C 180,E1 -25110,E2 -25110} C_VEL
LIN {X 0,Y 130.794,Z 696.172,A -85,B 0,C 180,E1 -25116.169,E2 -25116.169} C_VEL
LIN {X 0,Y 132.149,Z 693.945,A -85,B 0,C 180,E1 -25122.282,E2 -25122.282} C_VEL
LIN {X 0,Y 134.347,Z 691.109,A -85,B 0,C 180,E1 -25126.721,E2 -25126.721} C_VEL
LIN {X 0,Y 137.124,Z 687.274,A -85,B 0,C 180,E1 -25131.024,E2 -25131.024} C_VEL
LIN {X 0,Y 140.355,Z 682.184,A -85,B 0,C 180,E1 -25135.347,E2 -25135.347} C_VEL
LIN {X 0,Y 144.072,Z 676.141,A -85,B 0,C 180,E1 -25139.196,E2 -25139.196} C_VEL
LIN {X 0,Y 148.433,Z 668.349,A -85,B 0,C 180,E1 -25142.99,E2 -25142.99} C_VEL
LIN {X 0,Y 153.138,Z 658.665,A -85,B 0,C 180,E1 -25146.627,E2 -25146.627} C_VEL
LIN {X 0,Y 157.007,Z 649.605,A -85,B 0,C 180,E1 -25149.216,E2 -25149.216} C_VEL
LIN {X 0,Y 161.382,Z 638.038,A -85,B 0,C 180,E1 -25151.687,E2 -25151.687} C_VEL
LIN {X 0,Y 164.811,Z 626.389,A -85,B 0,C 180,E1 -25153.629,E2 -25153.629} C_VEL
LIN {X 0,Y 167.568,Z 614.566,A -85,B 0,C 180,E1 -25155.051,E2 -25155.051} C_VEL
LIN {X 0,Y 169.378,Z 601.695,A -85,B 0,C 180,E1 -25156.268,E2 -25156.268} C_VEL
LIN {X 0,Y 170.408,Z 589.245,A -85,B 0,C 180,E1 -25157.025,E2 -25157.025} C_VEL
LIN {X 0,Y 171.381,Z 569.238,A -85,B 0,C 180,E1 -25157.904,E2 -25157.904} C_VEL
LIN {X 0,Y 166.756,Z 559.898,A -85,B 0,C 180,E1 -25160.385,E2 -25160.385} C_VEL
LIN {X 0,Y 161.293,Z 550.274,A -85,B 0,C 180,E1 -25163.598,E2 -25163.598} C_VEL
LIN {X 0,Y 156.462,Z 542.734,A -85,B 0,C 180,E1 -25166.795,E2 -25166.795} C_VEL
LIN {X 0,Y 153.484,Z 538.452,A -85,B 0,C 180,E1 -25168.993,E2 -25168.993} C_VEL
LIN {X 0,Y 150.914,Z 534.705,A -85,B 0,C 180,E1 -25171.096,E2 -25171.096} C_VEL
LIN {X 0,Y 147.988,Z 530.733,A -85,B 0,C 180,E1 -25173.752,E2 -25173.752} C_VEL
LIN {X 0,Y 145.382,Z 527.696,A -85,B 0,C 180,E1 -25176.401,E2 -25176.401} C_VEL
LIN {X 0,Y 144.16,Z 525.747,A -85,B 0,C 180,E1 -25177.858,E2 -25177.858} C_VEL
LIN {X 0,Y 141.703,Z 523.434,A -85,B 0,C 180,E1 -25180.958,E2 -25180.958} C_VEL
LIN {X 0,Y 140.119,Z 520.469,A -85,B 0,C 180,E1 -25183.612,E2 -25183.612} C_VEL
LIN {X 0,Y 137.213,Z 518.216,A -85,B 0,C 180,E1 -25189.582,E2 -25189.582} C_VEL
LIN {X 0,Y 135.802,Z 515.211,A -85,B 0,C 180,E1 -25197.033,E2 -25197.033} C_VEL
LIN {X 0,Y 135.797,Z 514.736,A -85,B 0,C 180,E1 -25200,E2 -25200} C_VEL
LIN {X 0,Y 136.023,Z 515.855,A -85,B 0,C 180,E1 -25203.332,E2 -25203.332} C_VEL
LIN {X 0,Y 139.512,Z 520.207,A -85,B 0,C 180,E1 -25213.473,E2 -25213.473} C_VEL
LIN {X 0,Y 141.148,Z 522.587,A -85,B 0,C 180,E1 -25216.265,E2 -25216.265} C_VEL
LIN {X 0,Y 146.178,Z 531.051,A -85,B 0,C 180,E1 -25222.807,E2 -25222.807} C_VEL
LIN {X 0,Y 150.073,Z 538.025,A -85,B 0,C 180,E1 -25226.697,E2 -25226.697} C_VEL
LIN {X 0,Y 153.619,Z 544.867,A -85,B 0,C 180,E1 -25229.742,E2 -25229.742} C_VEL
LIN {X 0,Y 156.481,Z 550.674,A -85,B 0,C 180,E1 -25231.947,E2 -25231.947} C_VEL
LIN {X 0,Y 160.493,Z 559.458,A -85,B 0,C 180,E1 -25234.762,E2 -25234.762} C_VEL
LIN {X 0,Y 164.009,Z 568.304,A -85,B 0,C 180,E1 -25237.056,E2 -25237.056} C_VEL
LIN {X 0,Y 166.489,Z 575.374,A -85,B 0,C 180,E1 -25238.606,E2 -25238.606} C_VEL
LIN {X 0,Y 167.547,Z 604.208,A -85,B 0,C 180,E1 -25240.89,E2 -25240.89} C_VEL
LIN {X 0,Y 167.787,Z 618.874,A -85,B 0,C 180,E1 -25241.893,E2 -25241.893} C_VEL
LIN {X 0,Y 166.438,Z 632.085,A -85,B 0,C 180,E1 -25242.483,E2 -25242.483} C_VEL
LIN {X 0,Y 164.035,Z 645.502,A -85,B 0,C 180,E1 -25243.476,E2 -25243.476} C_VEL
LIN {X 0,Y 160.96,Z 657.827,A -85,B 0,C 180,E1 -25244.805,E2 -25244.805} C_VEL
LIN {X 0,Y 157.048,Z 669.68,A -85,B 0,C 180,E1 -25246.526,E2 -25246.526} C_VEL
LIN {X 0,Y 152.771,Z 680.348,A -85,B 0,C 180,E1 -25248.602,E2 -25248.602} C_VEL
LIN {X 0,Y 148.184,Z 690.111,A -85,B 0,C 180,E1 -25251.068,E2 -25251.068} C_VEL
LIN {X 0,Y 143.596,Z 699.052,A -85,B 0,C 180,E1 -25254.034,E2 -25254.034} C_VEL
LIN {X 0,Y 138.802,Z 707.825,A -85,B 0,C 180,E1 -25257.884,E2 -25257.884} C_VEL
LIN {X 0,Y 134.833,Z 714.897,A -85,B 0,C 180,E1 -25262.024,E2 -25262.024} C_VEL
LIN {X 0,Y 131.534,Z 720.593,A -85,B 0,C 180,E1 -25266.377,E2 -25266.377} C_VEL
LIN {X 0,Y 129.375,Z 725.152,A -85,B 0,C 180,E1 -25270.978,E2 -25270.978} C_VEL
LIN {X 0,Y 128.128,Z 728.652,A -85,B 0,C 180,E1 -25275.71,E2 -25275.71} C_VEL
LIN {X 0,Y 127.853,Z 731.655,A -85,B 0,C 180,E1 -25281.67,E2 -25281.67} C_VEL
LIN {X 0,Y 128.529,Z 733.088,A -85,B 0,C 180,E1 -25286.866,E2 -25286.866} C_VEL
LIN {X 0,Y 129.205,Z 733.417,A -85,B 0,C 180,E1 -25290,E2 -25290} C_VEL
LIN {X 0,Y 128.539,Z 733.074,A -85,B 0,C 180,E1 -25293.134,E2 -25293.134} C_VEL
LIN {X 0,Y 127.834,Z 731.152,A -85,B 0,C 180,E1 -25299.493,E2 -25299.493} C_VEL
LIN {X 0,Y 128.13,Z 728.597,A -85,B 0,C 180,E1 -25304.289,E2 -25304.289} C_VEL
LIN {X 0,Y 129.391,Z 725.072,A -85,B 0,C 180,E1 -25309.019,E2 -25309.019} C_VEL
LIN {X 0,Y 131.604,Z 720.495,A -85,B 0,C 180,E1 -25313.61,E2 -25313.61} C_VEL
LIN {X 0,Y 132.583,Z 718.716,A -85,B 0,C 180,E1 -25315.098,E2 -25315.098} C_VEL
LIN {X 0,Y 133.588,Z 715.879,A -85,B 0,C 180,E1 -25317.282,E2 -25317.282} C_VEL
LIN {X 0,Y 133.789,Z 710.77,A -85,B 0,C 180,E1 -25320.934,E2 -25320.934} C_VEL
LIN {X 0,Y 134.375,Z 705.12,A -85,B 0,C 180,E1 -25324.411,E2 -25324.411} C_VEL
LIN {X 0,Y 135.921,Z 701.383,A -85,B 0,C 180,E1 -25326.236,E2 -25326.236} C_VEL
LIN {X 0,Y 140.731,Z 692.646,A -85,B 0,C 180,E1 -25329.547,E2 -25329.547} C_VEL
LIN {X 0,Y 145.89,Z 682.551,A -85,B 0,C 180,E1 -25332.408,E2 -25332.408} C_VEL
LIN {X 0,Y 150.292,Z 672.595,A -85,B 0,C 180,E1 -25334.541,E2 -25334.541} C_VEL
LIN {X 0,Y 154.225,Z 661.776,A -85,B 0,C 180,E1 -25336.336,E2 -25336.336} C_VEL
LIN {X 0,Y 157.766,Z 649.913,A -85,B 0,C 180,E1 -25337.781,E2 -25337.781} C_VEL
LIN {X 0,Y 160.614,Z 636.886,A -85,B 0,C 180,E1 -25338.931,E2 -25338.931} C_VEL
LIN {X 0,Y 162.386,Z 624.445,A -85,B 0,C 180,E1 -25339.641,E2 -25339.641} C_VEL
LIN {X 0,Y 162.823,Z 617.185,A -85,B 0,C 180,E1 -25339.998,E2 -25339.998} C_VEL
LIN {X 0,Y 162.162,Z 585.258,A -85,B 0,C 180,E1 -25342.437,E2 -25342.437} C_VEL
LIN {X 0,Y 161.788,Z 577.598,A -85,B 0,C 180,E1 -25343.143,E2 -25343.143} C_VEL
LIN {X 0,Y 158.018,Z 567.033,A -85,B 0,C 180,E1 -25345.744,E2 -25345.744} C_VEL
LIN {X 0,Y 153.956,Z 557.432,A -85,B 0,C 180,E1 -25348.754,E2 -25348.754} C_VEL
LIN {X 0,Y 151.494,Z 552.041,A -85,B 0,C 180,E1 -25350.754,E2 -25350.754} C_VEL
LIN {X 0,Y 149.119,Z 547.233,A -85,B 0,C 180,E1 -25352.834,E2 -25352.834} C_VEL
LIN {X 0,Y 146.596,Z 542.128,A -85,B 0,C 180,E1 -25355.292,E2 -25355.292} C_VEL
LIN {X 0,Y 143.267,Z 535.861,A -85,B 0,C 180,E1 -25359.02,E2 -25359.02} C_VEL
LIN {X 0,Y 139.144,Z 528.509,A -85,B 0,C 180,E1 -25364.998,E2 -25364.998} C_VEL
LIN {X 0,Y 138.175,Z 527.021,A -85,B 0,C 180,E1 -25366.769,E2 -25366.769} C_VEL
LIN {X 0,Y 135.066,Z 523.137,A -85,B 0,C 180,E1 -25375.337,E2 -25375.337} C_VEL
LIN {X 0,Y 134.698,Z 521.795,A -85,B 0,C 180,E1 -25378.505,E2 -25378.505} C_VEL
LIN {X 0,Y 134.622,Z 521.531,A -85,B 0,C 180,E1 -25380,E2 -25380} C_VEL
LIN {X 0,Y 134.843,Z 522.545,A -85,B 0,C 180,E1 -25385.233,E2 -25385.233} C_VEL
LIN {X 0,Y 137.704,Z 526.768,A -85,B 0,C 180,E1 -25394.407,E2 -25394.407} C_VEL
LIN {X 0,Y 138.818,Z 527.495,A -85,B 0,C 180,E1 -25396.357,E2 -25396.357} C_VEL
LIN {X 0,Y 140.807,Z 530.931,A -85,B 0,C 180,E1 -25399.619,E2 -25399.619} C_VEL
LIN {X 0,Y 142.804,Z 532.878,A -85,B 0,C 180,E1 -25402.136,E2 -25402.136} C_VEL
LIN {X 0,Y 145.079,Z 536.3,A -85,B 0,C 180,E1 -25404.767,E2 -25404.767} C_VEL
LIN {X 0,Y 146.469,Z 537.927,A -85,B 0,C 180,E1 -25406.158,E2 -25406.158} C_VEL
LIN {X 0,Y 149.722,Z 542.607,A -85,B 0,C 180,E1 -25409.161,E2 -25409.161} C_VEL
LIN {X 0,Y 154.237,Z 549.32,A -85,B 0,C 180,E1 -25412.739,E2 -25412.739} C_VEL
LIN {X 0,Y 159.915,Z 558.916,A -85,B 0,C 180,E1 -25416.622,E2 -25416.622} C_VEL
LIN {X 0,Y 164.909,Z 568.481,A -85,B 0,C 180,E1 -25419.636,E2 -25419.636} C_VEL
LIN {X 0,Y 166.476,Z 572.1,A -85,B 0,C 180,E1 -25420.547,E2 -25420.547} C_VEL
LIN {X 0,Y 165.006,Z 596.994,A -85,B 0,C 180,E1 -25421.722,E2 -25421.722} C_VEL
LIN {X 0,Y 163.263,Z 610.398,A -85,B 0,C 180,E1 -25422.76,E2 -25422.76} C_VEL
LIN {X 0,Y 160.847,Z 622.492,A -85,B 0,C 180,E1 -25424.118,E2 -25424.118} C_VEL
LIN {X 0,Y 157.718,Z 633.831,A -85,B 0,C 180,E1 -25425.812,E2 -25425.812} C_VEL
LIN {X 0,Y 154.101,Z 643.995,A -85,B 0,C 180,E1 -25427.726,E2 -25427.726} C_VEL
LIN {X 0,Y 149.844,Z 654.303,A -85,B 0,C 180,E1 -25430.281,E2 -25430.281} C_VEL
LIN {X 0,Y 145.87,Z 662.704,A -85,B 0,C 180,E1 -25432.97,E2 -25432.97} C_VEL
LIN {X 0,Y 141.814,Z 670.423,A -85,B 0,C 180,E1 -25436.116,E2 -25436.116} C_VEL
LIN {X 0,Y 137.221,Z 678.082,A -85,B 0,C 180,E1 -25440.128,E2 -25440.128} C_VEL
LIN {X 0,Y 132.797,Z 684.877,A -85,B 0,C 180,E1 -25444.952,E2 -25444.952} C_VEL
LIN {X 0,Y 129.504,Z 689.481,A -85,B 0,C 180,E1 -25449.345,E2 -25449.345} C_VEL
LIN {X 0,Y 126.736,Z 693.015,A -85,B 0,C 180,E1 -25453.903,E2 -25453.903} C_VEL
